(* CODESYS project AlphaController_RECOVERED_2020-08-18T09-54-29.project
   Company: Sharp Packaging
   VersionPostfix: -alpha/pro24
   Version: 0.9.13.2
   Title: MOAB Prototype
   Author: Ben Hess

Project tree, tasks and I/O mapping:
  Device : Advantech Control x86 RTE V3, Advantech Co., Ltd., order no. 
      , version 3.5.13.0
    application Application
      libraries: Standard, * (System); VisuDialogs, * (System); Unit Conversion Interfaces, * (Intern); Festo_Motion_FHPP_3, 3.5.7.21 (Festo AG & Co. KG); Serial Communication, 3.5.7.0 (3S - Smart Software Solutions GmbH); Storage, 3.5.7.0 (3S - Smart Software Solutions GmbH); SysPort, 3.5.5.0 (System); Time and Date, 3.5.7.0 (3S - Smart Software Solutions GmbH); SysTime, 3.5.9.0 (System); Network, 3.5.7.0 (3S - Smart Software Solutions GmbH); CIP Object, * (3S - Smart Software Solutions GmbH); CAA Memory Block Manager Extern, * (CAA Technical Workgroup); CmpBitmapPool, * (System); IoDrvModbusBase, 3.5.13.0 (3S - Smart Software Solutions GmbH); SysFile, 3.5.15.0 (System); SysCom, 3.5.15.0 (System); Recipe Management, 3.5.15.0 (System); IoDrvModbus, 3.5.15.0 (3S - Smart Software Solutions GmbH); SysTypes Interfaces, * (System); BASIC, * (OSCAT)
      task IOUpdate (cyclic, interval 5 ms, priority 1) calls nothing
      task MainTask (cyclic, interval 5 ms, priority 0) calls PRG_MainProgram
      Event Handlers/
        function StartDone [ST]
        function OnlineChangeDone [ST]
        function PrepareShutdown [ST]
        function PrepareOnlineChange [ST]
        function PrepareStop [ST]
      Interfaces/
        interface IFaultHandler: AddActiveFault, RemoveActiveFault
        interface IComponentStatus: Mode, Ready
        interface ISupervisor: NotifyMachineFaulted, MakeReady
      RecipeManager
        recipe definition Recipes: HMIData.initiateCycle : BOOL; HMIData.ackAllFaults : BOOL; HMIData.makeReady : BOOL; HMIData.jobLoaded : BOOL; HMIData.stopMachine : BOOL; HMIData.version : STRING; HMIData.inCycle : BOOL; HMIData.batchEnable : BOOL; HMIData.batchSetting : UDINT; HMIData.batchCount : UDINT; HMIData.headCycleCount : UDINT; HMIData.pressureBarOpenDelay : REAL; HMIData.pressureBarCloseDelay : REAL; HMIData.passthroughSetting : REAL; HMIData.passthroughOffset : REAL; HMIData.passthroughPosition : REAL; HMIData.lpaDwell : REAL; HMIData.hpaDwell : REAL; HMIData.sealBarDwell : REAL; HMIData.sealBarTemperatureSetting : UDINT; HMIData.sealBarTemperature : UDINT; HMIData.sealFlattenersPosition : REAL; HMIData.bagSkirtLength : REAL; HMIData.bagLength : REAL; HMIData.bagWidth : REAL; HMIData.bagThickness : REAL; HMIData.bagTensionSetting : REAL; HMIData.bagDropTime : REAL; HMIData.bagForwardSpeed : UDINT; HMIData.bagReverseSpeed : UDINT; HMIData.bagEdgePhotoeyeCovered : BOOL; HMIData.printSpeed : UDINT; HMIData.printLength : REAL; HMIData.printOffset : REAL; HMIData.fillerCountSetting : UDINT; HMIData.fillerCurrentCount : UDINT; HMIData.fillerDropTime : REAL; HMIData.loadPlateDelay : REAL; HMIData.loadPlateDwell : REAL; HMIData.exitConveyorDwell : REAL; HMIData.vacuumDwell : REAL; HMIData.IBDDeflateDwellTime : REAL; HMIData.IBDPackageEjectAssistDelayTime : REAL; HMIData.IBDPackageEjectAssistDwellTime : REAL; HMIData.funnelInUse : BOOL; HMIData.funnelOpenDelay : REAL; HMIData.funnelOpeningTime : REAL; HMIData.funnelClosingTime : REAL; HMIData.externalExitConveyorDwell : REAL; HMIData.barcodeGoodReadCount : UDINT; HMIData.barcodeBadReadCount : UDINT; HMIData.barcodeBadReadFaultSetting : UDINT; HMIData.barcodeStartPosition : REAL; HMIData.barcodeScanDistance : REAL; HMIData.barcodeVerifierInUse : BOOL; HMIData.barcodeLastReadString : STRING(100); HMIData.lastCycleTime : REAL; HMIData.averageCycleTime : REAL; HMIData.resetAverageCycleTime : BOOL; HMIData.bagOpenRetrySetting : INT; HMIData.bagOpenRetryCount : INT; HMIData.bagOpenFeedNewBagSetting : INT; HMIData.bagOpenFeedNewBagCount : INT; HMIData.currentJobID : INT; HMIData.separateBeforeSeal : BOOL; HMIData.activateDemoMode : BOOL; HMIData.printerInUse : BOOL; HMIData.printerInstalled : BOOL; HMIData.lpaDuringBagFeedEnable : BOOL; HMIData.lpaBagEjectAssistEnable : BOOL; HMIData.lpaServiceOn : BOOL; HMIData.lpaServiceOff : BOOL; HMIData.lpaServicePulse : BOOL; HMIData.hpaServiceOn : BOOL; HMIData.hpaServicePulse : BOOL; HMIData.exitConveyorStart : BOOL; HMIData.exitConveyorStop : BOOL; HMIData.exitConveyorJog : BOOL; HMIData.exitConveyorJogTime : TIME; HMIData.exitConveyorStartDwell : BOOL; HMIData.pressureBarService.extendCommand : BOOL; HMIData.pressureBarService.retractCommand : BOOL; HMIData.pressureBarService.exhaustCommand : BOOL; HMIData.pressureBarService.extendedFeedback : BOOL; HMIData.pressureBarService.retractedFeedback : BOOL; HMIData.loadPlateService.extendCommand : BOOL; HMIData.loadPlateService.retractCommand : BOOL; HMIData.loadPlateService.exhaustCommand : BOOL; HMIData.loadPlateService.extendedFeedback : BOOL; HMIData.loadPlateService.retractedFeedback : BOOL; HMIData.forwardLoadPlateService.extendCommand : BOOL; HMIData.forwardLoadPlateService.retractCommand : BOOL; HMIData.forwardLoadPlateService.exhaustCommand : BOOL; HMIData.forwardLoadPlateService.extendedFeedback : BOOL; HMIData.forwardLoadPlateService.retractedFeedback : BOOL; HMIData.rearLoadPlateService.extendCommand : BOOL; HMIData.rearLoadPlateService.retractCommand : BOOL; HMIData.rearLoadPlateService.exhaustCommand : BOOL; HMIData.rearLoadPlateService.extendedFeedback : BOOL; HMIData.rearLoadPlateService.retractedFeedback : BOOL; HMIData.loadShelfService.extendCommand : BOOL; HMIData.loadShelfService.retractCommand : BOOL; HMIData.loadShelfService.exhaustCommand : BOOL; HMIData.loadShelfService.extendedFeedback : BOOL; HMIData.loadShelfService.retractedFeedback : BOOL; HMIData.IBDService.extendCommand : BOOL; HMIData.IBDService.retractCommand : BOOL; HMIData.IBDService.exhaustCommand : BOOL; HMIData.IBDService.extendedFeedback : BOOL; HMIData.IBDService.retractedFeedback : BOOL; HMIData.funnelService.extendCommand : BOOL; HMIData.funnelService.retractCommand : BOOL; HMIData.funnelService.exhaustCommand : BOOL; HMIData.funnelService.extendedFeedback : BOOL; HMIData.funnelService.retractedFeedback : BOOL; HMIData.jogBagForward : BOOL; HMIData.jogBagReverse : BOOL; HMIData.jogPassthroughForward : BOOL; HMIData.jogPassthroughReverse : BOOL; HMIData.sealBarServiceCycle : BOOL; HMIData.sealBarServiceRetract : BOOL; HMIData.sealBarServiceExtend : BOOL; HMIData.bagOpenFingersServiceGrab : BOOL; HMIData.bagOpenFingersServiceRelease : BOOL; HMIData.sealFlattenersServiceRaise : BOOL; HMIData.sealFlattenersServiceLower : BOOL; HMIData.sealFlattenersServiceJogIn : BOOL; HMIData.sealFlattenersServiceJogOut : BOOL; HMIData.sealFlattenersManualPositionSetting : REAL; HMIData.sealFlattenersMoveToManualPos : BOOL; HMIData.passthroughManualPositionSetting : REAL; HMIData.passthroughMoveToManualPos : BOOL; HMIData.factoryTestMode : BOOL; HMIData.vacuumServiceOn : BOOL; HMIData.vacuumServiceOff : BOOL; HMIData.printHeadServiceRaise : BOOL; HMIData.printHeadServiceLower : BOOL; HMIData.externalExitConveyorStart : BOOL; HMIData.externalExitConveyorStop : BOOL; HMIData.externalExitConveyorJog : BOOL; HMIData.externalExitConveyorStartDwell : BOOL; HMIData.triggerBarcodeReaderService : BOOL; HMIData.bofSelection : INT; HMIData.sealFlattenersSelection : INT; HMIData.printerSelection : INT; HMIData.integratedExitConveyorSelection : INT; HMIData.externalExitConveyorSelection : INT; HMIData.packageEjectSelection : INT; HMIData.independentBagDeflatorSelection : INT; HMIData.cycleStartButtonSelection : INT; HMIData.barcodeVerifierSelection : INT; HMIData.baggerModelSelection : INT; HMIData.auxIOConfig.factorySelection : INT; HMIData.auxIOConfig.cfgInputSelection : INT; HMIData.auxIOConfig.cfgOutput1Selection : INT; HMIData.auxIOConfig.cfgOutput2Selection : INT; HMIData.fillerFactorySelection : INT; HMIData.funnelFactorySelection : INT; HMIData.murrIOConfigVersion : INT; HMIData.printerConfigVersion : INT; HMIData.frontFilmFeedMotorConfigVersion : INT; HMIData.rearUnwindMotorConfigVersion : INT; HMIData.sealFlattenerMotorConfigVersion : INT; HMIData.printerRibbonLow.active : BOOL; HMIData.printerNotReady.active : BOOL; HMIData.waitingForPrinter.active : BOOL; HMIData.sealBarNotAtTemperature.active : BOOL; HMIData.recoveryModeActive.active : BOOL; HMIData.jobLoadRequired.active : BOOL; HMIData.baggerNotReady.active : BOOL; HMIData.demoModeIsActive.active : BOOL; HMIData.factoryTestModeActive.active : BOOL; HMIData.machineNotTested.active : BOOL; HMIData.packageEjectGuardRemoved.active : BOOL; HMIData.bagLevelLow.active : BOOL; HMIData.fillerModeCycleStartOnly.active : BOOL; HMIData.baggerInhibited.active : BOOL; HMIData.pressureBarState : STRING; HMIData.baggerCycles.reset : BOOL; HMIData.baggerCycles.count : UDINT; HMIData.bagOpenFingerCycles.reset : BOOL; HMIData.bagOpenFingerCycles.count : UDINT; HMIData.bagsMade.reset : BOOL; HMIData.bagsMade.count : UDINT; HMIData.sealBarCycles.reset : BOOL; HMIData.sealBarCycles.count : UDINT; HMIData.pressureBarCycles.reset : BOOL; HMIData.pressureBarCycles.count : UDINT; HMIData.passthroughChanges.reset : BOOL; HMIData.passthroughChanges.count : UDINT; HMIData.loadPlateCycles.reset : BOOL; HMIData.loadPlateCycles.count : UDINT; HMIData.printerCycles.reset : BOOL; HMIData.printerCycles.count : UDINT; HMIData.motorizedSealFlattenerCycles.reset : BOOL; HMIData.motorizedSealFlattenerCycles.count : UDINT; HMIData.bagOpenRetryTotal.reset : BOOL; HMIData.bagOpenRetryTotal.count : UDINT; HMIData.bagsRejectedTotal.reset : BOOL; HMIData.bagsRejectedTotal.count : UDINT; HMIData.resettableBagsMade.reset : BOOL; HMIData.resettableBagsMade.count : UDINT; HMIData.airFilterClean.target : UDINT; HMIData.airFilterClean.name : STRING; HMIData.airFilterClean.units : STRING; HMIData.airFilterClean.reset : BOOL; HMIData.airFilterClean.count : UDINT; HMIData.driveRollerClean.target : UDINT; HMIData.driveRollerClean.name : STRING; HMIData.driveRollerClean.units : STRING; HMIData.driveRollerClean.reset : BOOL; HMIData.driveRollerClean.count : UDINT; HMIData.printHeadClean.target : UDINT; HMIData.printHeadClean.name : STRING; HMIData.printHeadClean.units : STRING; HMIData.printHeadClean.reset : BOOL; HMIData.printHeadClean.count : UDINT; HMIData.pressureBarGuideShaftGuides.target : UDINT; HMIData.pressureBarGuideShaftGuides.name : STRING; HMIData.pressureBarGuideShaftGuides.units : STRING; HMIData.pressureBarGuideShaftGuides.reset : BOOL; HMIData.pressureBarGuideShaftGuides.count : UDINT; HMIData.pressureBarLeak.iExtended : BOOL; HMIData.pressureBarLeak.iRetracted : BOOL; HMIData.pressureBarLeak.maximumStrokeTime : REAL; HMIData.pressureBarLeak.strokeTime : REAL; HMIData.pressureBarLeak.strokeTimer.IN : BOOL; HMIData.pressureBarLeak.strokeTimer.PT : TIME; HMIData.pressureBarLeak.strokeTimer.Q : BOOL; HMIData.pressureBarLeak.strokeTimer.ET : TIME; HMIData.pressureBarLeak.extendedONS.CLK : BOOL; HMIData.pressureBarLeak.extendedONS.Q : BOOL; HMIData.pressureBarLeak.retractedONS.CLK : BOOL; HMIData.pressureBarLeak.retractedONS.Q : BOOL; HMIData.pressureBarLeak.target : UDINT; HMIData.pressureBarLeak.name : STRING; HMIData.pressureBarLeak.units : STRING; HMIData.pressureBarLeak.reset : BOOL; HMIData.pressureBarLeak.count : UDINT; HMIData.loadPlateLeak.iExtended : BOOL; HMIData.loadPlateLeak.iRetracted : BOOL; HMIData.loadPlateLeak.maximumStrokeTime : REAL; HMIData.loadPlateLeak.strokeTime : REAL; HMIData.loadPlateLeak.strokeTimer.IN : BOOL; HMIData.loadPlateLeak.strokeTimer.PT : TIME; HMIData.loadPlateLeak.strokeTimer.Q : BOOL; HMIData.loadPlateLeak.strokeTimer.ET : TIME; HMIData.loadPlateLeak.extendedONS.CLK : BOOL; HMIData.loadPlateLeak.extendedONS.Q : BOOL; HMIData.loadPlateLeak.retractedONS.CLK : BOOL; HMIData.loadPlateLeak.retractedONS.Q : BOOL; HMIData.loadPlateLeak.target : UDINT; HMIData.loadPlateLeak.name : STRING; HMIData.loadPlateLeak.units : STRING; HMIData.loadPlateLeak.reset : BOOL; HMIData.loadPlateLeak.count : UDINT; HMIData.msfHorizontalMotorTemp.iDriveTemp : DINT; HMIData.msfHorizontalMotorTemp.maxTemp : REAL; HMIData.msfHorizontalMotorTemp.DriveTemp : REAL; HMIData.msfHorizontalMotorTemp.target : UDINT; HMIData.msfHorizontalMotorTemp.name : STRING; HMIData.msfHorizontalMotorTemp.units : STRING; HMIData.msfHorizontalMotorTemp.reset : BOOL; HMIData.msfHorizontalMotorTemp.count : UDINT; HMIData.bagDeliveryMotorTemp.iDriveTemp : DINT; HMIData.bagDeliveryMotorTemp.maxTemp : REAL; HMIData.bagDeliveryMotorTemp.DriveTemp : REAL; HMIData.bagDeliveryMotorTemp.target : UDINT; HMIData.bagDeliveryMotorTemp.name : STRING; HMIData.bagDeliveryMotorTemp.units : STRING; HMIData.bagDeliveryMotorTemp.reset : BOOL; HMIData.bagDeliveryMotorTemp.count : UDINT; HMIData.passthroughMotorTemp.iDriveTemp : DINT; HMIData.passthroughMotorTemp.maxTemp : REAL; HMIData.passthroughMotorTemp.DriveTemp : REAL; HMIData.passthroughMotorTemp.target : UDINT; HMIData.passthroughMotorTemp.name : STRING; HMIData.passthroughMotorTemp.units : STRING; HMIData.passthroughMotorTemp.reset : BOOL; HMIData.passthroughMotorTemp.count : UDINT; HMIData.faultActive : BOOL
      Types/
        data type DEVICE_MODES
        Factoy Selection/
          data type IntegratedConveyorSelection
          data type LabelPrinterSelection
          data type PackageEjectionSelection
          data type ExteralConveyorSelection
          data type BCVSelection
          data type BagDeflatorSelection
          data type SealFlattenerSelection
          data type PalmButtonSelection
          data type BagOpenFingersSelection
          data type AuxiliaryIOSelection
          data type FillerSelection
          data type ModelSelection
          data type FunnelSelection
        data type MODBUS_COMM_TYPE
        data type LoadPlateFaultsType
        data type MotorCommFault
        data type Fault
        data type QX_PROGRAMS
        data type PRINT_SPEEDS
        States/
          data type SOLENOID_TEST_STATES
          data type AMP_EIP_MOVE_INITIAL_STATES
          data type MOVE_MODBUS_COMMAND_STATES
          data type JOG_STATES
          data type PRESSURE_BAR_STATES
          data type VACUUM_PICKER_STATES
          data type OPCODE_MODBUS_COMMAND_STATES
          data type FILLER_STATES
          data type GRABBER_STATES
          data type BCR_STATES
          data type PASSTHROUGH_SERVO_STATES
          Head/
            data type TEST_HEAD_STATES
            data type PRINTER_STATES
            data type HEAD_STATES
            data type SEAL_FLATTENER_STATES
            data type SEAL_BAR_STATES
            data type SEAL_SEPARATE_STATES
            data type FINISH_CYCLE_STATES
            data type RELEASE_FEED_STATES
            data type BAG_DELIVERY_STATES
            data type BAG_OPEN_ASSIST_STATES
          MurrIOMOdule/
            data type MOM_STATES
            data type MURR_SYSTEM_STATES
          data type JAW_HOMING_STATES
        HMI Types/
          data type PressureBarHMI
        data type ServiceCommands
        data type ORIENTAL_OPERATION_TYPES
        data type PressureBarFaultsType
        data type IOMasterFaultsType
        data type CylinderFaultsType
        data type ModbusLongType
        AuxIO/
          data type AuxOutputSelection
          data type AuxInputSelection
          data type AuxIOConfiguration
        data type Alarm
        data type FaultType
        data type Warning
        data type StepServoFaultsType
        data type STEP_SERVO_OPCODES
        data type CONFIG_VERSIONS
      global variables HMIData
      trace Trace (task MainTask): PRG_Bagger.moabHead.pressureBar.electricPressureBarMotor.CRTL_Axis.AckStart, PRG_Bagger.moabHead.pressureBar.electricPressureBarMotor.CRTL_Axis.StartTask, PRG_Bagger.moabHead.pressureBar.electricPressureBarMotor.CRTL_Axis.ActualRecordNo, PRG_Bagger.moabHead.pressureBar.electricPressureBarMotor.CRTL_Axis.RecordNo
      FBs/
        DataHandlers/
          function block FB_ModbusDWORD [ST]: HighWord, RawValue, LowWord
          function block ModbusLongHandlerFB [ST]: PackDirect, Pack, Unpack
        Fault/
          function block FB_ONS [ST]
          function block FB_GetTime [ST]
          function block FB_Fault [ST]: Execute, InstanceName, RegisterLogger, Ack, Trigger, FB_Init
          data type LogMessageType
          function block FB_HMIFault [ST]: FB_Init, FB_Reinit, Initialize, InstanceName, Execute
          function block FB_InternalLogger [ST]: InstanceName, AddLogItem
        function block FB_TCPClient [ST]: SendLabel
        Cylinders/
          function block FB_CylinderWithFeedback [ST]: Execute
          interface IThreePositonCylinder: Exhaust
          function block FB_CylinderFaults [ST]
          function block FB_Cylinder [ST]: Retract, Extend, Execute
          function block FB_ThreePositionCylinderWithFeedback [ST]: ResetFault, Exhaust, Execute, Faulted
          interface ICylinder: Extend, Execute, Retract
          function block FB_ThreePositionCylinder [ST]: Exhaust
        function block FB_WriteToFile [ST]
        function block FB_PredictiveMaint [ST]
        function block GetTime [ST]
        function block FB_CylinderLeak [ST]
        function block FB_DriveTemp [ST]
        function block TimeLeftFB [ST]
        Components/
          function block PrinterFB_Mode2 [ST]: AutoSendPrintSignal, AutoPrintNow, AutoAckPrintDone, Ready, Mode
          function block BagDeliveryFB_BothMotors [ST]: Ready, ClearCommands, Mode, AutoReverseBag, AutoPrinterDone, AutoWaitForPrinter, AutoStartPrintFeed, AutoFeedBagOut, AutoFeedToEye, AutoPrinterReady
          KeyenceL20FB/
            data type eKeyenceLN20_Error_ID
            function block KeyenceNL20FB [ST]: Ready, Mode
            data type eKeyenceLN20FB_States
          function block MotorizedSealFlattenersFB_BagFeed [ST]: AutoMoveIn, AutoMoveToBagHolding, AutoMoveToHandLoad, Ready, Mode, ClearCommands, AutoMoveToClearance, AutoMoveOut
          function block BarcodeReaderFB [ST]: Trigger, BadRead, GoodRead
          function block BagDeliveryFB [ST]: AutoPrinterDone, AutoFeedToEye, AutoWaitForPrinter, AutoReverseBag, ClearCommands, AutoPrinterReady, Mode, Ready, AutoFeedBagOut, AutoStartPrintFeed
          function block AdjustablePassthroughFB [ST]: MovePassthrough, Ready, Mode, AckRequest, HomeEndStop
          function block FillerFB [ST]: BaggerCycledAndReady, Ready, BaggerCycleInitiated, Mode, Reset
          function block PrinterFB [ST]: AutoSendPrintSignal, AutoPrintNow, Mode, AutoAckPrintDone, Ready
          DelayDwellFB/
            function block DelayDwellFB [ST]: Reset, ManualOff, ManualOn, Trigger, DwellSetting, DelaySetting
            data type DELAY_DWELL_STATES
          FB_MotorizedPressureBar/
            function block FB_CylinderFeedback [ST]
            function block FB_MotorizedPressureBar [ST]: CloseJawNoLatch, CloseJaw, OpenJaw, HomeNow
            data type MotorizedPbarStates
          function block BagOpenFingersFB [ST]: Release, Grab
          function block MotorizedSealFlattenersFB [ST]: ClearCommands, AutoMoveOut, Mode, Ready, AutoMoveToClearance, AutoMoveToBagHolding, AutoMoveIn
          function block PneumaticPressureBarFB_1 [ST]: AutoSealBag, RetractCylinder, AutoOpenJaw, ExhaustCylinder, AutoDoneMovingPassthrough, Mode, ExtendCylinderHighPressure, AutoCloseJaw, Ready, AutoMovingPassthrough, ExtendCylinderLowPressure
          function block FunnelFB [ST]: DelaySetting, CloseNow, OpeningTime, OpenNow, ClosingTime
          FB_MotorizedIBD/
            data type MotorizedIBDStates
            function block FB_MotorizedIBD [ST]: CloseIBD, OpenFull, OpenIBD, RemovePower, HomeNow
          function block PneumaticPressureBarFB [ST]: AutoDoneMovingPassthrough, AutoMovingPassthrough, ExhaustCylinder, Ready, Mode, AutoCloseJaw, ExtendCylinderHighPressure, ExtendCylinderLowPressure, AutoOpenJaw, RetractCylinder, AutoSealBag
          function block ElectricPressureBarFB [ST]: AutoCloseJaw, AutoOpenJaw, Mode, Ready, ClearCommands
          function block PickAndPlaceFB [ST]
          function block BagOpenFingersWithSensorsFB [ST]: CheckIfBagGrabbed
          function block MurrIOFB [ST]: Mode, Ready
          function block BaseComponentFB [ST]: Ready, Reset, Mode
          function block HeadRaiseLowerFB [ST]
          function block MonostableMultivibratorFB [ST]: DelaySetting, Trigger, ManualOn, ManualOff, DwellSetting
        Motors/
          interface IPositionableMotor: Homing, Moving, InPosition, CurrentPosition, Stop, CommandAcknowledged, HomeNow, MoveToPosition, HomeRequired, MoveDistance
          interface IStoredProgramMotor: ActiveStoredProgramNumber, ExecuteStoredProgram
          Applied Motion/
            function block FB_AppliedMotionBagDeliveryMotor_1 [ST]: SetRearMotorToTorqueMode, SetRearMotorToEncoderFollowing, MoveDistance, StopViaProgram, CommandAcknowledged, SetTorque, Execute, SetRearMotorTorqueValue, MoveDistanceFinal
            Modbus Commands/
              function block FB_SendUserRegistersAppliedMotionTCP [ST]: Execute
              function block FB_SendMoveCommandAppliedMotionRTU [ST]: Execute, CheckIfParSendSuccessful
              function block FB_SendBagMoveAppliedMotionTCP [ST]: Execute
              function block FB_SendMoveCommandAppliedMotionTCP [ST]: Execute
              function block FB_SendOpcodeCommandAppliedMotionTCP [ST]: Execute
              function block FB_SendOpcodeCommandAppliedMotionRTU [ST]: Execute
            function block FB_AppliedMotionStepServoMBBase [ST]: Execute, HomeRequired, CommandAcknowledged, ExecuteStoredProgram, ActiveStoredProgramNumber, MoveDistance, InPosition, HomeNow, Stop, Homing, CurrentPosition, Moving, MoveToPosition
            function block FB_AppliedMotionStepServoEIPPassthrough [ST]: HomeNow, DoneClamping, AllowClamping, Stop, SetPositionLimit, Execute
            DataHandlers/
              function block FB_StepServoAlarms [ST]
              function block FB_StepServoCommands [ST]: Enable, AlarmReset, SendHostCommand, FeedToLength, Clear, StopNormal, IdleState, Disable, StopCrash, SendQAndExecute, FeedToPosition
              function block StepServoStatusFB [ST]
            function block FB_AppliedMotionStepServoEIPPassthrough_1 [ST]: DoneClamping, AllowClamping
            function block FB_AppliedMotionBagDeliveryMotorNoFollowing [ST]: MoveDistance, SetRearMotorToTorqueMode, Execute, SetRearMotorToEncoderFollowing, MoveDistanceFinal, CommandAcknowledged, StopViaProgram
            function block FB_AppliedMotionStepServoTCP [ST]: Stop, MoveToPosition, ExecuteStoredProgram, MoveDistance, HomeNow
            function block FB_AppliedMotionStepServoEIPBase [ST]: Stop, Homing, HomeNow, MoveDistance, CommandAcknowledged, InstanceName, MachineFaulted, MoveToPositionTorque, InPosition, Disable, Enable, ResetEncoderPosition, Execute, HomeRequired, ActiveStoredProgramNumber, Reset, Faulted, MoveToPosition, SetTorque, ExecuteStoredProgram, CurrentPosition, Moving, MoveDistanceTorque
            function block FB_AppliedMotionBagDeliveryMotor [ST]: MoveDistance, SendParameters, MoveDistanceFinal, StopViaProgram
            function block FB_AppliedMotionStepServoEIPBaseQX [ST]: Execute, CommandAcknowledged, HomeNow, HomeRequired, Moving, ActiveStoredProgramNumber, InPosition, MoveDistanceTorque, MachineFaulted, Faulted, MoveToPosition, MoveToPositionTorque, Stop, MoveDistance, CurrentPosition, Homing, Reset, RegisterWithFaultHandler, ExecuteStoredProgram
          Festo/
            function block FB_FestoMotor [ST]: ExecuteStoredProgram, Homing, HomeRequired, CurrentPosition, Execute, CommandAcknowledged, Stop, ActiveStoredProgramNumber, InitDrive, Moving, MoveDistance, InPosition, MoveToPosition, HomeNow
        Temp Sensors/
          function block FB_TemperatureSensor [ST]: TempReadingC, TempReadingF, InstanceName
          function block FB_IFMTempSensor [ST]: Execute
          function block FB_TempController [ST]
          interface ITempSensor: TempReadingF, TempReadingC
        function block FB_HMILight [ST]: BlinkSlow, BlinkFast, TurnOff, TurnOn
        function block FB_FaultHandler [ST]: registerFaultSource
        function block SerialMotorTestFB [ST]
        function block FB_BaggerHeadRaise [ST]
        FunctionalAreas/
          function block FB_MOABHead_Electric [ST]
          function block FB_MOABHead [ST]
        function block FB_CycleCounter [ST]: Increment, Clear, SetCount
      Programs/
        program PRG_Bagger [ST]
        program Faults [ST]
        function block PRG_ [ST]
        program PRG_MainProgram [ST]
      global variables Globals
      function SaveValues [ST]
      Symbols
      ObjectHandling/
        interface IExecuteAutomatically: Execute
        function block FB_CollectionHandlerAll [ST]: AddObject
        interface IResettable
        interface IFault: Trigger, Ack
        function block FB_CollectionHandlerLogs [ST]: AddObject
        function block FB_CollectionHandlerLoggable [ST]: RegisterAll, AddObject
        interface IAllObjects: InstanceName
        function block FB_CollectionHandlerInitializable [ST]: InitializeAll, AddObject
        global variables GlobalObjects
        function block FB_CollectionHandlerActiveFaults [ST]: RemoveObject, AckAll, AddObject
        interface ILoggable: RegisterLogger
        interface IInitializable: Initialize
        interface IExhaustable
        interface IFault_1: Ack, Trigger
        function block FB_CollectionHandlerFaults [ST]: AckAll, AddObject
        interface IMachineLogger: AddLogItem
        function block FB_CollectionHandlerExecutable [ST]: ExecuteAll, AddObject
      function RecallValues [ST]
    System_Diagnosis : System Diagnosis, Advantech Co., Ltd., version 3.5.13.0
        unmapped channels: System Information
    CIFX_EIP : CIFX-EIP, 3S - Smart Software Solutions GmbH, order no. 1, version 3.5.12.0
        settings: IPAddress = [16#C0,16#A8,16#0A,16#15]; SubnetMask = [16#FF,16#FF,16#FF,16#00]; GatewayAddress = [16#00,16#00,16#00,16#00]; ConfigVersion = 50660608
      IBD_Motor : SSM23IP-3EG, Applied Motion Products, Inc, order no. SSM23IP-3EG, version Major Revision=16#3, Minor Revision = 16#3
          settings: INITIALIZED = TRUE; IP address of Target = [16#C0,16#A8,16#0A,16#39]; MAC address of Target = [16#00,16#00,16#00,16#00,16#00,16#00]; Keying.Check Device Type = FALSE; Keying.Check Vendor Code = FALSE; Keying.Check Product Code = FALSE; Keying.Check Major Revision = FALSE; Keying.Check Minor Revision = FALSE; RequiredConfigVersion = 50660864; Number of Connections = 1; Connection Settings.Requested packet intervall = 10000 µs; Connection Settings.OT Connection Parameters = 18502; Connection Settings.TO Connection Parameters = 18490; Connection Settings.Connection Flags = 1056; Connection Settings.Connection Path Size = 8; Status Code.ReadOnly = False; Status Code.BitSize = 32; Status Code.DataSize = 4; Alarm Code.ReadOnly = False; Alarm Code.BitSize = 32; Alarm Code.DataSize = 4; Supply Voltage.ReadOnly = False; Supply Voltage.BitSize = 32; Supply Voltage.DataSize = 4; Actual Current.ReadOnly = False; Actual Current.BitSize = 32; Actual Current.DataSize = 4; Drive Temperature.ReadOnly = False; Drive Temperature.BitSize = 32; Drive Temperature.DataSize = 4; Encoder Position.ReadOnly = False; Encoder Position.BitSize = 32; Encoder Position.DataSize = 4; Absolute Position.ReadOnly = False; Absolute Position.BitSize = 32; Absolute Position.DataSize = 4; Position Error.ReadOnly = False; Position Error.BitSize = 32; Position Error.DataSize = 4; Actual Velocity.ReadOnly = False ... (246 more)
          input  iIBDMotorEIP : DINT  // Status Code
          output oIBDMotorEIP : DINT  // Command Word
          unmapped channels: Alarm Code, Supply Voltage, Actual Current, Drive Temperature, Encoder Position, Absolute Position, Position Error, Actual Velocity, Input Status (extended), Input Status (main), Output Status, Analog Input 1 ... (16 more)
      Cube67_BN_E_V2 : Cube67+ BN-E V2, Murrelektronik GmbH, order no. 56535, version Major Revision=16#2, Minor Revision = 16#5
          settings: INITIALIZED = TRUE; IP address of Target = [16#C0,16#A8,16#0A,16#64]; Keying.Check Vendor Code = FALSE; Keying.Check Product Code = FALSE; Keying.Check Major Revision = FALSE; Keying.Check Minor Revision = FALSE; RequiredConfigVersion = 50660864; Number of Connections = 1; Connection Settings.Requested packet intervall = 5000 µs; Connection Settings.OT Connection Parameters = 18624; Connection Settings.TO Connection Parameters = 18708; Connection Settings.Connection Flags = 1056; Connection Settings.Connection Path Size = 8; Input AssemblyParam0.ReadOnly = False; Input AssemblyParam0.BitSize = 8; Input AssemblyParam0.DataSize = 1; Input AssemblyParam1.ReadOnly = False; Input AssemblyParam1.BitSize = 8; Input AssemblyParam1.DataSize = 1; Input AssemblyParam2.ReadOnly = False; Input AssemblyParam2.BitSize = 8; Input AssemblyParam2.DataSize = 1; Input AssemblyParam3.ReadOnly = False; Input AssemblyParam3.BitSize = 8; Input AssemblyParam3.DataSize = 1; Input AssemblyParam4.ReadOnly = False; Input AssemblyParam4.BitSize = 8; Input AssemblyParam4.DataSize = 1; Input AssemblyParam5.ReadOnly = False; Input AssemblyParam5.BitSize = 8; Input AssemblyParam5.DataSize = 1; Input AssemblyParam6.ReadOnly = False; Input AssemblyParam6.BitSize = 8; Input AssemblyParam6.DataSize = 1; Input AssemblyParam7.ReadOnly = False; Input AssemblyParam7.BitSize = 8; Input AssemblyParam7.DataSize = 1; Input AssemblyParam8.ReadOnly = False; Input AssemblyParam8.BitSize = 8; Input AssemblyParam8.DataSize = 1 ... (4114 more)
          input  iAuxFillerTrigger : BOOL  // Input AssemblyParam29.Bit0
          input  iAuxFillerOK : BOOL  // Input AssemblyParam29.Bit1
          input  iAuxConfigInput : BOOL  // Input AssemblyParam29.Bit2
          input  iFunnelOpened : BOOL  // Input AssemblyParam30.Bit0
          input  iRightPalmButton : BOOL  // Input AssemblyParam30.Bit3
          input  iFunnelClosed : BOOL  // Input AssemblyParam31.Bit0
          input  iLeftPalmButton : BOOL  // Input AssemblyParam31.Bit3
          input  iLoadPlateRetracted : BOOL  // Input AssemblyParam32.Bit0
          input  iLoadShelfRetracted : BOOL  // Input AssemblyParam32.Bit1
          input  iEStopOK : BOOL  // Input AssemblyParam32.Bit2
          input  iFrontLoadPlateRetracted : BOOL  // Input AssemblyParam32.Bit3
          input  iHeadLowered : BOOL  // Input AssemblyParam32.Bit6
          input  iLoadPlateExtended : BOOL  // Input AssemblyParam33.Bit0
          input  iLoadShelfExtended : BOOL  // Input AssemblyParam33.Bit1
          input  iFrontLoadPlateExtended : BOOL  // Input AssemblyParam33.Bit3
          input  iBagsLow : BOOL  // Input AssemblyParam33.Bit5
          input  iHeadRaised : BOOL  // Input AssemblyParam33.Bit6
          input  printerDataReady : BOOL  // Input AssemblyParam35.Bit0
          input  printerEndOfPrint : BOOL  // Input AssemblyParam35.Bit1
          input  printerReady : BOOL  // Input AssemblyParam35.Bit2
          input  iPrinterRibbonEncoder : BOOL  // Input AssemblyParam35.Bit3
          input  iBarcodeReadGood : BOOL  // Input AssemblyParam35.Bit4
          input  iJawClampsExtended : BOOL  // Input AssemblyParam36.Bit0
          input  iLefttFingerBagPresent : BOOL  // Input AssemblyParam36.Bit2
          input  iJawClampsRetracted : BOOL  // Input AssemblyParam37.Bit0
          input  iPressureBarNotObstructed : BOOL  // Input AssemblyParam37.Bit1
          input  iRightFingerBagPresent : BOOL  // Input AssemblyParam37.Bit2
          input  iPowerOffButton : BOOL  // Input AssemblyParam37.Bit3
          input  iHeaterBarTempInputs : BYTE  // Input AssemblyParam38
          input  iMurrSystemState : BYTE  // Input Assembly_Param200
          output oMOMConfig : BYTE  // Output AssemblyParam0
          output oAuxBaggerOK : BOOL  // Output Assembly_Param28.Bit0
          output oAuxConfigOut1 : BOOL  // Output Assembly_Param28.Bit1
          output oAuxReadyForFiller : BOOL  // Output Assembly_Param28.Bit2
          output oAuxConfigOut2 : BOOL  // Output Assembly_Param28.Bit3
          output oSoftStart : BOOL  // Output Assembly_Param32.Bit4
          output oBaggerHeadMotorDir : BOOL  // Output Assembly_Param32.Bit7
          output oRunExitConveyor : BOOL  // Output Assembly_Param33.Bit2
          output oRunBaggerHeadMotor : BOOL  // Output Assembly_Param33.Bit7
          output oPrinterStartPrint : BOOL  // Output Assembly_Param34.Bit0
          output oRunPrinterRibbonUnwindMotor : BOOL  // Output Assembly_Param34.Bit1
          output oBarcodeTrigger : BOOL  // Output Assembly_Param34.Bit2
          output oRunExternalExitConveyor : BOOL  // Output Assembly_Param36.Bit1
          output oHMILight : BOOL  // Output Assembly_Param36.Bit3
          output oHeaterPulse : BOOL  // Output Assembly_Param37.Bit4
          unmapped channels: Input AssemblyParam0, Input AssemblyParam1, Input AssemblyParam2, Input AssemblyParam3, Input AssemblyParam4, Input AssemblyParam5, Input AssemblyParam6, Input AssemblyParam7, Input AssemblyParam8, Input AssemblyParam9, Input AssemblyParam10, Input AssemblyParam11 ... (445 more)
      MSFMotor : SSM23IP-3EG, Applied Motion Products, Inc, order no. SSM23IP-3EG, version Major Revision=16#3, Minor Revision = 16#3
          settings: INITIALIZED = TRUE; IP address of Target = [16#C0,16#A8,16#0A,16#35]; Keying.Check Device Type = FALSE; Keying.Check Vendor Code = FALSE; Keying.Check Product Code = FALSE; Keying.Check Major Revision = FALSE; Keying.Check Minor Revision = FALSE; RequiredConfigVersion = 50660864; Number of Connections = 1; Connection Settings.Requested packet intervall = 5000 µs; Connection Settings.OT Connection Parameters = 18502; Connection Settings.TO Connection Parameters = 18490; Connection Settings.Connection Flags = 1056; Connection Settings.Connection Path Size = 8; Status Code.ReadOnly = False; Status Code.BitSize = 32; Status Code.DataSize = 4; Alarm Code.ReadOnly = False; Alarm Code.BitSize = 32; Alarm Code.DataSize = 4; Supply Voltage.ReadOnly = False; Supply Voltage.BitSize = 32; Supply Voltage.DataSize = 4; Actual Current.ReadOnly = False; Actual Current.BitSize = 32; Actual Current.DataSize = 4; Drive Temperature.ReadOnly = False; Drive Temperature.BitSize = 32; Drive Temperature.DataSize = 4; Encoder Position.ReadOnly = False; Encoder Position.BitSize = 32; Encoder Position.DataSize = 4; Absolute Position.ReadOnly = False; Absolute Position.BitSize = 32; Absolute Position.DataSize = 4; Position Error.ReadOnly = False; Position Error.BitSize = 32; Position Error.DataSize = 4; Actual Velocity.ReadOnly = False; Actual Velocity.BitSize = 32 ... (245 more)
          input  sealFlattenerHorizontalMotorInputs : DINT  // Status Code
          output sealFlattenerHorizontalMotorOutputs : DINT  // Command Word
          unmapped channels: Alarm Code, Supply Voltage, Actual Current, Drive Temperature, Encoder Position, Absolute Position, Position Error, Actual Velocity, Input Status (extended), Input Status (main), Output Status, Analog Input 1 ... (16 more)
      Bag_Delivery_Rear_Motor : TSM34IP, Applied Motion Products, Inc, order no. TSM34IP, version Major Revision=16#3, Minor Revision = 16#3
          settings: INITIALIZED = TRUE; IP address of Target = [16#C0,16#A8,16#0A,16#38]; MAC address of Target = [16#00,16#00,16#00,16#00,16#00,16#00]; Keying.Check Device Type = FALSE; Keying.Check Vendor Code = FALSE; Keying.Check Product Code = FALSE; Keying.Check Major Revision = FALSE; Keying.Check Minor Revision = FALSE; RequiredConfigVersion = 50660864; Number of Connections = 1; Connection Settings.Requested packet intervall = 10000 µs; Connection Settings.OT Connection Parameters = 18502; Connection Settings.TO Connection Parameters = 18490; Connection Settings.Connection Flags = 1056; Connection Settings.Connection Path Size = 8; Status Code.ReadOnly = False; Status Code.BitSize = 32; Status Code.DataSize = 4; Alarm Code.ReadOnly = False; Alarm Code.BitSize = 32; Alarm Code.DataSize = 4; Supply Voltage.ReadOnly = False; Supply Voltage.BitSize = 32; Supply Voltage.DataSize = 4; Actual Current.ReadOnly = False; Actual Current.BitSize = 32; Actual Current.DataSize = 4; Drive Temperature.ReadOnly = False; Drive Temperature.BitSize = 32; Drive Temperature.DataSize = 4; Encoder Position.ReadOnly = False; Encoder Position.BitSize = 32; Encoder Position.DataSize = 4; Absolute Position.ReadOnly = False; Absolute Position.BitSize = 32; Absolute Position.DataSize = 4; Position Error.ReadOnly = False; Position Error.BitSize = 32; Position Error.DataSize = 4; Actual Velocity.ReadOnly = False ... (246 more)
          input  bagRearMotorInputs AT %ID200 : DINT  // Status Code
          input  iBagTensionFault : BOOL  // Output Status.Bit3
          output bagRearMotorOutputs AT %QD200 : DINT  // Command Word
          unmapped channels: Alarm Code, Supply Voltage, Actual Current, Drive Temperature, Encoder Position, Absolute Position, Position Error, Actual Velocity, Input Status (extended), Input Status (main), Output Status, Analog Input 1 ... (16 more)
      FestoManifold : CTEU-EP EtherNetIP bus node, Festo AG & Co. KG, order no. CTEU-EP, version Major Revision=16#2, Minor Revision = 16#2
          settings: INITIALIZED = TRUE; IP address of Target = [16#C0,16#A8,16#0A,16#6E]; Keying.Check Vendor Code = FALSE; Keying.Check Product Code = FALSE; Keying.Check Major Revision = FALSE; Keying.Check Minor Revision = FALSE; RequiredConfigVersion = 50660864; Number of Connections = 1; Connection Settings.Requested packet intervall = 10000 µs; Connection Settings.OT Connection Parameters = 18446; Connection Settings.TO Connection Parameters = 18442; Connection Settings.Connection Flags = 1056; Connection Settings.Connection Path Size = 8; Connection Settings.Config#2 Size = 38; Single Port Inputs 8 bytesParam8.ReadOnly = False; Single Port Inputs 8 bytesParam8.BitSize = 8; Single Port Inputs 8 bytesParam8.DataSize = 1; Single Port Inputs 8 bytesParam9.ReadOnly = False; Single Port Inputs 8 bytesParam9.BitSize = 8; Single Port Inputs 8 bytesParam9.DataSize = 1; Single Port Inputs 8 bytesParam10.ReadOnly = False; Single Port Inputs 8 bytesParam10.BitSize = 8; Single Port Inputs 8 bytesParam10.DataSize = 1; Single Port Inputs 8 bytesParam11.ReadOnly = False; Single Port Inputs 8 bytesParam11.BitSize = 8; Single Port Inputs 8 bytesParam11.DataSize = 1; Single Port Inputs 8 bytesParam12.ReadOnly = False; Single Port Inputs 8 bytesParam12.BitSize = 8; Single Port Inputs 8 bytesParam12.DataSize = 1; Single Port Inputs 8 bytesParam13.ReadOnly = False; Single Port Inputs 8 bytesParam13.BitSize = 8; Single Port Inputs 8 bytesParam13.DataSize = 1; Single Port Inputs 8 bytesParam14.ReadOnly = False; Single Port Inputs 8 bytesParam14.BitSize = 8; Single Port Inputs 8 bytesParam14.DataSize = 1; Single Port Inputs 8 bytesParam15.ReadOnly = False; Single Port Inputs 8 bytesParam15.BitSize = 8; Single Port Inputs 8 bytesParam15.DataSize = 1; Single Port Outputs 8bytesParam8.ReadOnly = False; Single Port Outputs 8bytesParam8.BitSize = 8 ... (119 more)
          output oJawClampExtend : BOOL  // Single Port Outputs 8bytesParam8.Bit0
          output oJawClampRetract : BOOL  // Single Port Outputs 8bytesParam8.Bit1
          output oSealBarExtend : BOOL  // Single Port Outputs 8bytesParam8.Bit2
          output oSealBarRetract : BOOL  // Single Port Outputs 8bytesParam8.Bit3
          output oLPAOn : BOOL  // Single Port Outputs 8bytesParam8.Bit4
          output oHPAOn : BOOL  // Single Port Outputs 8bytesParam8.Bit5
          output oLoadPlateExtend : BOOL  // Single Port Outputs 8bytesParam8.Bit6
          output oLoadPlateRetract : BOOL  // Single Port Outputs 8bytesParam8.Bit7
          output oBOFUp : BOOL  // Single Port Outputs 8bytesParam9.Bit0
          output oBOFDown : BOOL  // Single Port Outputs 8bytesParam9.Bit1
          output oPrintHeadDown : BOOL  // Single Port Outputs 8bytesParam9.Bit2
          output oPrintHeadUp : BOOL  // Single Port Outputs 8bytesParam9.Bit3
          output oVacOn : BOOL  // Single Port Outputs 8bytesParam9.Bit4
          output oSealFlatUp : BOOL  // Single Port Outputs 8bytesParam9.Bit6
          output oSealFlatDown : BOOL  // Single Port Outputs 8bytesParam9.Bit7
          output oFrontLoadPlateToLoad : BOOL  // Single Port Outputs 8bytesParam10.Bit2
          output oLoadShelfUp : BOOL  // Single Port Outputs 8bytesParam10.Bit4
          output oIBDExtend : BOOL  // Single Port Outputs 8bytesParam10.Bit6
          output oIBDRetract : BOOL  // Single Port Outputs 8bytesParam10.Bit7
          output oFunnelOpen : BOOL  // Single Port Outputs 8bytesParam11.Bit0
          output oFunnelClose : BOOL  // Single Port Outputs 8bytesParam11.Bit1
          unmapped channels: Single Port Inputs 8 bytesParam8, Single Port Inputs 8 bytesParam9, Single Port Inputs 8 bytesParam10, Single Port Inputs 8 bytesParam11, Single Port Inputs 8 bytesParam12, Single Port Inputs 8 bytesParam13, Single Port Inputs 8 bytesParam14, Single Port Inputs 8 bytesParam15, Single Port Outputs 8bytesParam8, Single Port Outputs 8bytesParam9, Single Port Outputs 8bytesParam10, Single Port Outputs 8bytesParam11 ... (4 more)
      Pbar_ServoEIP : SSM23IP-3EG, Applied Motion Products, Inc, order no. SSM23IP-3EG, version Major Revision=16#3, Minor Revision = 16#3
          settings: INITIALIZED = TRUE; IP address of Target = [16#C0,16#A8,16#0A,16#34]; Keying.Check Vendor Code = FALSE; Keying.Check Product Code = FALSE; Keying.Check Major Revision = FALSE; Keying.Check Minor Revision = FALSE; RequiredConfigVersion = 50660864; Number of Connections = 1; Connection Settings.Requested packet intervall = 5000 µs; Connection Settings.OT Connection Parameters = 18502; Connection Settings.TO Connection Parameters = 18490; Connection Settings.Connection Flags = 1056; Connection Settings.Connection Path Size = 8; Status Code.ReadOnly = False; Status Code.BitSize = 32; Status Code.DataSize = 4; Alarm Code.ReadOnly = False; Alarm Code.BitSize = 32; Alarm Code.DataSize = 4; Supply Voltage.ReadOnly = False; Supply Voltage.BitSize = 32; Supply Voltage.DataSize = 4; Actual Current.ReadOnly = False; Actual Current.BitSize = 32; Actual Current.DataSize = 4; Drive Temperature.ReadOnly = False; Drive Temperature.BitSize = 32; Drive Temperature.DataSize = 4; Encoder Position.ReadOnly = False; Encoder Position.BitSize = 32; Encoder Position.DataSize = 4; Absolute Position.ReadOnly = False; Absolute Position.BitSize = 32; Absolute Position.DataSize = 4; Position Error.ReadOnly = False; Position Error.BitSize = 32; Position Error.DataSize = 4; Actual Velocity.ReadOnly = False; Actual Velocity.BitSize = 32; Actual Velocity.DataSize = 4 ... (244 more)
          input  jawPasstrhoughMotorInputs : DINT  // Status Code
          input  iJawClamped : BOOL  // Input Status (main).Bit1
          input  iJawClearToClamp : BOOL  // Input Status (main).Bit2
          output jawPasstrhoughMotorOutputs : DINT  // Command Word
          unmapped channels: Alarm Code, Supply Voltage, Actual Current, Drive Temperature, Encoder Position, Absolute Position, Position Error, Actual Velocity, Input Status (extended), Input Status (main), Output Status, Analog Input 1 ... (16 more)
      Keyence_BCV : Generic EtherNet/IP device, 3S - Smart Software Solutions GmbH, version 3.5.15.0
          settings: INITIALIZED = TRUE; IP address of Target = [16#C0,16#A8,16#0A,16#A1]; MAC address of Target = [16#00,16#00,16#00,16#00,16#00,16#00]; Keying.Compatibility Bit = FALSE; RequiredConfigVersion = 50660864; Number of Connections = 1; Connection Settings.Requested packet intervall (µs) = 10000; Connection Settings.OT Connection Parameters = 18514; Connection Settings.TO Connection Parameters = 18606; Connection Settings.Connection Flags = 1056; Connection Settings.Connection Path Size = 8; Connection Path = [16#20,16#04,16#24,16#01,16#2C,16#65,16#2C,16#64]; Input_Param0.ReadOnly = False; Input_Param0.BitSize = 8; Input_Param0.DataSize = 1; Input_Param1.ReadOnly = False; Input_Param1.BitSize = 8; Input_Param1.DataSize = 1; Input_Param2.ReadOnly = False; Input_Param2.BitSize = 8; Input_Param2.DataSize = 1; Input_Param3.ReadOnly = False; Input_Param3.BitSize = 8; Input_Param3.DataSize = 1; Input_Param4.ReadOnly = False; Input_Param4.BitSize = 8; Input_Param4.DataSize = 1; Input_Param5.ReadOnly = False; Input_Param5.BitSize = 8; Input_Param5.DataSize = 1; Input_Param6.ReadOnly = False; Input_Param6.BitSize = 8; Input_Param6.DataSize = 1; Input_Param7.ReadOnly = False; Input_Param7.BitSize = 8; Input_Param7.DataSize = 1; Input_Param8.ReadOnly = False; Input_Param8.BitSize = 8; Input_Param8.DataSize = 1; Input_Param9.ReadOnly = False ... (2205 more)
          input  keyenceBCVInputs : BYTE  // Input_Param0
          output keyenceBCVOutputs : BYTE  // Output_Param0
          unmapped channels: Input_Param1, Input_Param2, Input_Param3, Input_Param4, Input_Param5, Input_Param6, Input_Param7, Input_Param8, Input_Param9, Input_Param10, Input_Param11, Input_Param12 ... (234 more)
      Bag_Delivery_EIP_Motor : TSM34IP, Applied Motion Products, Inc, order no. TSM34IP, version Major Revision=16#3, Minor Revision = 16#3
          settings: INITIALIZED = TRUE; IP address of Target = [16#C0,16#A8,16#0A,16#37]; Keying.Check Vendor Code = FALSE; Keying.Check Product Code = FALSE; Keying.Check Major Revision = FALSE; Keying.Check Minor Revision = FALSE; RequiredConfigVersion = 50660864; Number of Connections = 1; Connection Settings.Requested packet intervall = 5000 µs; Connection Settings.OT Connection Parameters = 18502; Connection Settings.TO Connection Parameters = 18490; Connection Settings.Connection Flags = 1056; Connection Settings.Connection Path Size = 8; Status Code.ReadOnly = False; Status Code.BitSize = 32; Status Code.DataSize = 4; Alarm Code.ReadOnly = False; Alarm Code.BitSize = 32; Alarm Code.DataSize = 4; Supply Voltage.ReadOnly = False; Supply Voltage.BitSize = 32; Supply Voltage.DataSize = 4; Actual Current.ReadOnly = False; Actual Current.BitSize = 32; Actual Current.DataSize = 4; Drive Temperature.ReadOnly = False; Drive Temperature.BitSize = 32; Drive Temperature.DataSize = 4; Encoder Position.ReadOnly = False; Encoder Position.BitSize = 32; Encoder Position.DataSize = 4; Absolute Position.ReadOnly = False; Absolute Position.BitSize = 32; Absolute Position.DataSize = 4; Position Error.ReadOnly = False; Position Error.BitSize = 32; Position Error.DataSize = 4; Actual Velocity.ReadOnly = False; Actual Velocity.BitSize = 32; Actual Velocity.DataSize = 4 ... (244 more)
          input  bagDeliveryMotorInputs : DINT  // Status Code
          input  iBagNotPresent : BOOL  // Input Status (main).Bit2
          output bagDeliveryMotorOutputs : DINT  // Command Word
          unmapped channels: Alarm Code, Supply Voltage, Actual Current, Drive Temperature, Encoder Position, Absolute Position, Position Error, Actual Velocity, Input Status (extended), Input Status (main), Output Status, Analog Input 1 ... (16 more)
    Ethernet : Ethernet, 3S - Smart Software Solutions GmbH, version 3.5.15.0
        settings: IPAddress = [192,168,10,20]; SubnetMask = [255,255,255,0]; GatewayAddress = [192,168,10,254]; MACAddress = [16#74,16#FE,16#48,16#3F,16#C0,16#65]; NetworkInterfaceName = 'Machine LAN:2'; NetworkInterfaceName = "Machine LAN:2"; SaveCommunicationSettings = FALSE
      Modbus_TCP_Master : Modbus TCP Master, 3S - Smart Software Solutions GmbH, version 3.5.15.0 (disabled)
          settings: AutoReconnect = TRUE
        Bag_Delivery_Master_Motor : Modbus TCP Slave, 3S - Smart Software Solutions GmbH, version 3.5.15.0 (disabled)
            settings: Unit-ID = 255; IPAddress = [192, 168, 10, 55]; Read Registers.Function Code = 3; Read Registers.Read Offset = 16#0000; Read Registers.Read Length = 125; Read Registers.Write Offset = 0; Read Registers.Write Length = 0; Read Registers.Cycle Time = 50
            input  BagDeliverMasterMotorModbusInputs AT %IW536 : ARRAY[0..124] OF WORD  // Read Registers
        PBar_Servo : Modbus TCP Slave, 3S - Smart Software Solutions GmbH, version 3.5.15.0 (disabled)
            settings: Unit-ID = 255; ResponseTimeout = 100; IPAddress = [192, 168, 10, 52]; Channel 0.Function Code = 3; Channel 0.Read Offset = 16#0000; Channel 0.Read Length = 125; Channel 0.Write Offset = 0; Channel 0.Write Length = 0; Channel 0.Cycle Time = 100
            input  PressureBarEndStopTCPMotorModbusInputs AT %IW800 : ARRAY[0..124] OF WORD  // Channel 0
      EtherNet_IP_Scanner : EtherNet/IP Scanner, 3S - Smart Software Solutions GmbH, order no. 1, version 3.5.15.20
        AMP_Test_Motor : STM23IP-3EN, Applied Motion Products, Inc, order no. STM23IP-3EN, version Major Revision=16#3, Minor Revision = 16#3 (disabled)
            settings: INITIALIZED = TRUE; IP address of Target = [16#C0,16#A8,16#0A,16#37]; Keying.Check Vendor Code = FALSE; Keying.Check Product Code = FALSE; Keying.Check Major Revision = FALSE; Keying.Check Minor Revision = FALSE; RequiredConfigVersion = 50660864; Number of Connections = 1; Connection Settings.Requested packet intervall (µs) = 10000; Connection Settings.OT Connection Parameters = 18502; Connection Settings.TO Connection Parameters = 18490; Connection Settings.Connection Flags = 1056; Connection Settings.Connection Path Size = 8; Connection Path = [16#20,16#04,16#24,16#66,16#2C,16#70,16#2C,16#65]; Status Code.ReadOnly = False; Status Code.BitSize = 32; Status Code.DataSize = 4; Alarm Code.ReadOnly = False; Alarm Code.BitSize = 32; Alarm Code.DataSize = 4; Supply Voltage.ReadOnly = False; Supply Voltage.BitSize = 32; Supply Voltage.DataSize = 4; Actual Current.ReadOnly = False; Actual Current.BitSize = 32; Actual Current.DataSize = 4; Drive Temperature.ReadOnly = False; Drive Temperature.BitSize = 32; Drive Temperature.DataSize = 4; Encoder Position.ReadOnly = False; Encoder Position.BitSize = 32; Encoder Position.DataSize = 4; Absolute Position.ReadOnly = False; Absolute Position.BitSize = 32; Absolute Position.DataSize = 4; Position Error.ReadOnly = False; Position Error.BitSize = 32; Position Error.DataSize = 4; Actual Velocity.ReadOnly = False; Actual Velocity.BitSize = 32 ... (245 more)
            unmapped channels: Status Code, Alarm Code, Supply Voltage, Actual Current, Drive Temperature, Encoder Position, Absolute Position, Position Error, Actual Velocity, Input Status (extended), Input Status (main), Output Status ... (18 more)
        EX260_SEN1 : EX260-SEN1, SMC Corporation, order no. EX260-SEN1, version Major Revision=16#2, Minor Revision = 16#2 (disabled)
            settings: INITIALIZED = TRUE; IP address of Target = [16#C0,16#A8,16#0A,16#A2]; Keying.Check Minor Revision = FALSE; RequiredConfigVersion = 50660864; Number of Connections = 1; Connection Settings.Requested packet intervall (µs) = 20000; Connection Settings.OT Connection Parameters = 18442; Connection Settings.TO Connection Parameters = 18436; Connection Settings.Connection Flags = 1056; Connection Settings.Connection Path Size = 8; Connection Path = [16#20,16#04,16#24,16#69,16#2C,16#96,16#2C,16#64]; Output size.Name = Output size; Output size.ReadOnly = False; Output size.BitSize = 8; Output size.DataSize = 1; Output size.DataType = 'SINT'; Output size.ReadOnly = False; Output size.BitSize = 8; Output size.DataSize = 1; Input size.ReadOnly = False; Input size.BitSize = 16; Input size.DataSize = 1; Output Param0.ReadOnly = False; Output Param0.BitSize = 8; Output Param0.DataSize = 1; Output Param1.ReadOnly = False; Output Param1.BitSize = 8; Output Param1.DataSize = 1; Output Param2.ReadOnly = False; Output Param2.BitSize = 8; Output Param2.DataSize = 1; Output size.ReadOnly = False; Output size.BitSize = 8; Output size.DataSize = 1; Input size.Name = 'Input size'; Input size.HelpString = ''; Input size.ReadOnly = False; Input size.BitSize = 16; Input size.DataSize = 1; Input size.DataType = 'SINT' ... (25 more)
            output oExtendCylinder : BOOL  // Output Param0.Bit0
            output oRetractCylinder : BOOL  // Output Param0.Bit1
            output oExtendSealBar : BOOL  // Output Param0.Bit2
            output oPositionBagOpenFingersToRelease : BOOL  // Output Param0.Bit4
            output oMovePrintHeadDown : BOOL  // Output Param0.Bit6
            unmapped channels: %IB0 Input size, %QB0 Output Param0, %QB1 Output Param1, %QB2 Output Param2, %QB3 Output size
        PickAndPlaceY : STM23IP-3EN, Applied Motion Products, Inc, order no. STM23IP-3EN, version Major Revision=16#2, Minor Revision = 16#33 (disabled)
            settings: INITIALIZED = TRUE; IP address of Target = [16#C0,16#A8,16#0A,16#3B]; Keying.Check Device Type = FALSE; Keying.Check Vendor Code = FALSE; Keying.Check Product Code = FALSE; Keying.Check Major Revision = FALSE; Keying.Check Minor Revision = FALSE; RequiredConfigVersion = 50660864; Number of Connections = 1; Connection Settings.Requested packet intervall (µs) = 50000; Connection Settings.OT Connection Parameters = 18502; Connection Settings.TO Connection Parameters = 18490; Connection Settings.Connection Flags = 1056; Connection Settings.Connection Path Size = 8; Connection Settings.Config#1 Size = 2; Configuration Data = [16#0,16#0]; Connection Path = [16#20,16#04,16#24,16#66,16#2C,16#70,16#2C,16#65]; Status Code.ReadOnly = False; Status Code.BitSize = 32; Status Code.DataSize = 4; Alarm Code.ReadOnly = False; Alarm Code.BitSize = 32; Alarm Code.DataSize = 4; Supply Voltage.ReadOnly = False; Supply Voltage.BitSize = 32; Supply Voltage.DataSize = 4; Actual Current.ReadOnly = False; Actual Current.BitSize = 32; Actual Current.DataSize = 4; Drive Temperature.ReadOnly = False; Drive Temperature.BitSize = 32; Drive Temperature.DataSize = 4; Encoder Position.ReadOnly = False; Encoder Position.BitSize = 32; Encoder Position.DataSize = 4; Absolute Position.ReadOnly = False; Absolute Position.BitSize = 32; Absolute Position.DataSize = 4; Position Error.ReadOnly = False; Position Error.BitSize = 32 ... (248 more)
            input  pickAndPlaceYMotorInputs AT %ID117 : DINT  // Status Code
            output pickAndPlaceYMotorOutputs AT %QD97 : DINT  // Command Word
            unmapped channels: Alarm Code, Supply Voltage, Actual Current, Drive Temperature, Encoder Position, Absolute Position, Position Error, Actual Velocity, Input Status (extended), Input Status (main), Output Status, Analog Input 1 ... (16 more)
        PickAndPlaceX : STM23IP-3EN, Applied Motion Products, Inc, order no. STM23IP-3EN, version Major Revision=16#2, Minor Revision = 16#33 (disabled)
            settings: INITIALIZED = TRUE; IP address of Target = [16#C0,16#A8,16#0A,16#3A]; Keying.Check Device Type = FALSE; Keying.Check Vendor Code = FALSE; Keying.Check Product Code = FALSE; Keying.Check Major Revision = FALSE; Keying.Check Minor Revision = FALSE; RequiredConfigVersion = 50660864; Number of Connections = 1; Connection Settings.Requested packet intervall (µs) = 50000; Connection Settings.OT Connection Parameters = 18502; Connection Settings.TO Connection Parameters = 18490; Connection Settings.Connection Flags = 1056; Connection Settings.Connection Path Size = 8; Connection Settings.Config#1 Size = 2; Configuration Data = [16#0,16#0]; Connection Path = [16#20,16#04,16#24,16#66,16#2C,16#70,16#2C,16#65]; Status Code.ReadOnly = False; Status Code.BitSize = 32; Status Code.DataSize = 4; Alarm Code.ReadOnly = False; Alarm Code.BitSize = 32; Alarm Code.DataSize = 4; Supply Voltage.ReadOnly = False; Supply Voltage.BitSize = 32; Supply Voltage.DataSize = 4; Actual Current.ReadOnly = False; Actual Current.BitSize = 32; Actual Current.DataSize = 4; Drive Temperature.ReadOnly = False; Drive Temperature.BitSize = 32; Drive Temperature.DataSize = 4; Encoder Position.ReadOnly = False; Encoder Position.BitSize = 32; Encoder Position.DataSize = 4; Absolute Position.ReadOnly = False; Absolute Position.BitSize = 32; Absolute Position.DataSize = 4; Position Error.ReadOnly = False; Position Error.BitSize = 32 ... (248 more)
            input  pickAndPlaceXMotorInputs AT %ID103 : DINT  // Status Code
            output pickAndPlaceXMotorOutputs AT %QD81 : DINT  // Command Word
            unmapped channels: Alarm Code, Supply Voltage, Actual Current, Drive Temperature, Encoder Position, Absolute Position, Position Error, Actual Velocity, Input Status (extended), Input Status (main), Output Status, Analog Input 1 ... (16 more)
        PickAndPlaceZ : STM23IP-3EN, Applied Motion Products, Inc, order no. STM23IP-3EN, version Major Revision=16#2, Minor Revision = 16#33 (disabled)
            settings: INITIALIZED = TRUE; IP address of Target = [16#C0,16#A8,16#0A,16#3C]; Keying.Check Device Type = FALSE; Keying.Check Vendor Code = FALSE; Keying.Check Product Code = FALSE; Keying.Check Major Revision = FALSE; Keying.Check Minor Revision = FALSE; RequiredConfigVersion = 50660864; Number of Connections = 1; Connection Settings.Requested packet intervall (µs) = 30000; Connection Settings.OT Connection Parameters = 18502; Connection Settings.TO Connection Parameters = 18490; Connection Settings.Connection Flags = 1056; Connection Settings.Connection Path Size = 8; Connection Settings.Config#1 Size = 2; Configuration Data = [16#0,16#0]; Connection Path = [16#20,16#04,16#24,16#66,16#2C,16#70,16#2C,16#65]; Status Code.ReadOnly = False; Status Code.BitSize = 32; Status Code.DataSize = 4; Alarm Code.ReadOnly = False; Alarm Code.BitSize = 32; Alarm Code.DataSize = 4; Supply Voltage.ReadOnly = False; Supply Voltage.BitSize = 32; Supply Voltage.DataSize = 4; Actual Current.ReadOnly = False; Actual Current.BitSize = 32; Actual Current.DataSize = 4; Drive Temperature.ReadOnly = False; Drive Temperature.BitSize = 32; Drive Temperature.DataSize = 4; Encoder Position.ReadOnly = False; Encoder Position.BitSize = 32; Encoder Position.DataSize = 4; Absolute Position.ReadOnly = False; Absolute Position.BitSize = 32; Absolute Position.DataSize = 4; Position Error.ReadOnly = False; Position Error.BitSize = 32 ... (248 more)
            input  pickAndPlaceZMotorInputs AT %ID1 : DINT  // Status Code
            output pickAndPlaceZMotorOutputs AT %QD113 : DINT  // Command Word
            unmapped channels: Alarm Code, Supply Voltage, Actual Current, Drive Temperature, Encoder Position, Absolute Position, Position Error, Actual Velocity, Input Status (extended), Input Status (main), Output Status, Analog Input 1 ... (16 more)
  Project Information/
    function GetVersion [ST]
    function GetCompany [ST]
    function GetTitle [ST]
    function GetTextProperty2 [ST]
    function GetTextProperty [ST]
    function GetBooleanProperty [ST]
    function GetVersionProperty [ST]
    function GetNumberProperty [ST]
  text list GlobalTextList
  Library Information/
    function IsLibReleased [ST]
    function GetLibVersion [ST]
    function GetLibVersionNumber [ST]
  text list System
*)

// Device/Application/Types/States/Head/TEST_HEAD_STATES
{attribute 'qualified_only'}
{attribute 'strict'}
TYPE TEST_HEAD_STATES :
(
	Idle := 0,
	Cycling := 10,
	StartHoming := 20,
	Homing := 21,
	HomingComplete := 22,
	MovePassthrough := 30,
	MovingPassthrough := 31,
	MovedPassthrough := 32,
	Fault := 99
);
END_TYPE

// Device/Application/Types/DEVICE_MODES
{attribute 'qualified_only'}
{attribute 'strict'}
TYPE DEVICE_MODES :
(
	Manual := 0,	// Control only from service
	Auto := 1,		// Control only from main Bagger Program
	SemiAuto := 2	// Independent control (like as a test fixture)
);
END_TYPE

// Device/Application/Types/States/SOLENOID_TEST_STATES
{attribute 'qualified_only'}
{attribute 'strict'}
TYPE SOLENOID_TEST_STATES :
(
	Extended := 0,
	Retracted := 1,
	FailedToExtend := 2,
	Idle := 3
);
END_TYPE

// Device/Application/Types/Factoy Selection/IntegratedConveyorSelection
{attribute 'qualified_only'}
{attribute 'strict'}
TYPE IntegratedConveyorSelection :
(
	NotInstalled := 0,
	RearExit := 1
);
END_TYPE

// Device/Application/Types/States/Head/PRINTER_STATES
{attribute 'strict'}
{attribute 'qualified_only'}
TYPE PRINTER_STATES :
(
	Idle := 0,
	WaitingForData := 1,
	DataReady := 2,
	BeginPrintCycle := 3,	
	FeedAtPrintSpeed := 10,
	Printing := 11,
	DonePrinting := 20,
	FeedThrough := 21,
	Ready := 40,
	Fault := 99
);
END_TYPE

// Device/Application/Types/Factoy Selection/LabelPrinterSelection
{attribute 'qualified_only'}
{attribute 'strict'}
TYPE LabelPrinterSelection :
(
	NotInstalled := 0,
	ZebraPrinter203DPI := 1,
	ZebraPrinter300DPI := 2
);
END_TYPE

// Device/Application/Types/States/AMP_EIP_MOVE_INITIAL_STATES
{attribute 'strict'}
{attribute 'qualified_only'}
TYPE AMP_EIP_MOVE_INITIAL_STATES :
(
	Idle := 0,
	SetOutputOff := 10,
	WaitAfterSettingOutputOff := 11,
	MoveMotor := 12,
	WaitAfterMovingMotor := 13,
	SetOutputOn := 14,
	WaitAfterSettingOutputOn := 15,
	Fault := 99
);
END_TYPE

// Device/Application/Types/MODBUS_COMM_TYPE
{attribute 'strict'}
{attribute 'qualified_only'}
TYPE MODBUS_COMM_TYPE :
(
	ModbusTCP := 0,
	ModbusRTU := 1
);
END_TYPE

// Device/Application/Types/AuxIO/AuxOutputSelection
{attribute 'qualified_only'}
{attribute 'strict'}
TYPE AuxOutputSelection :
(
	NotConfigured := 0,
	PrinterDataReady := 1,
	WaitingForPrinter := 2,
	CycleComplete := 3,
	BagMade := 4,
	BagMadePlusLabelRequired := 5,
	BagsLow := 6
);
END_TYPE

// Device/Application/Types/LoadPlateFaultsType
TYPE LoadPlateFaultsType :
STRUCT
	failedToDischarge : FB_Fault(name := 'Failed to Discharge');        // Load Plate failed to reach Discharge Position
    failedToLoad : FB_Fault(name := 'Failed to Load');  // Load Plate failed to reach Loading Position
	sensorFault : FB_Fault(name := 'Failed to Sensor Fault');		// Both sensors active at the same time
END_STRUCT
END_TYPE

// Device/Application/Types/States/MOVE_MODBUS_COMMAND_STATES
{attribute 'strict'}
{attribute 'qualified_only'}
TYPE MOVE_MODBUS_COMMAND_STATES :
(
	Idle := 0,
	SendParameters := 10,
	WaitAfterParametersSent := 11,
	SendOpcode := 20,
	WaitAfterOpcodeSent := 21,
	SendCommand := 31,
	WaitAfterCommandSent := 32,
	SendClearCommand := 40,
	WaitAfterSendClearCommand := 41,
	Fault := 99
);
END_TYPE

// Device/Application/Types/MotorCommFault
TYPE MotorCommFault :
STRUCT
	timeOfFault : DATE_AND_TIME;
	message : STRING;
END_STRUCT
END_TYPE

// Device/Application/Types/Factoy Selection/PackageEjectionSelection
{attribute 'qualified_only'}
{attribute 'strict'}
TYPE PackageEjectionSelection :
(
	NotInstalled := 0,
	RearRetractingLoadPlate := 1,
	LabelSideUp := 2
);
END_TYPE

// Device/Application/Types/States/MurrIOMOdule/MOM_STATES
{attribute 'strict'}
{attribute 'qualified_only'}
TYPE MOM_STATES :
(
	Idle := 0,
	Reverse := 1,
	Reversing := 2,
	ReverseToPrinthead := 3,
	ReversingToPrintHead := 4,
	ReverseDone := 5,
	WaitingForPrinter := 10,
	FeedToPrintOffset := 11,
	FeedingToPrintOffset := 12,
	FedToPrintOffset := 13,
	FeedAtPrintSpeed := 20,
	FeedingAtPrintSpeed := 21,
	FedAtPrintSpeed := 22,
	FeedBagOut := 30,
	FeedingBagOut := 31,
	FedBagOut := 32,
	Ready := 40,
	FeedToEye := 50,
	FeedingToEye := 51,
	SetTorqueMode := 52,
	Fault := 99,
	Manual := 100
);
END_TYPE

// Device/Application/Types/States/JOG_STATES
{attribute 'strict'}
{attribute 'qualified_only'}
TYPE JOG_STATES :
(
    Idle := 0,
    JogForwardDIRequest := 10,
    JogForwardOpcodeRequest := 11,
    JoggingForward := 12,
    JogReverseDIRequest := 20,
    JogReverseOpcodeRequest := 21,
    JoggingReverse := 22,
    StoppingJog := 30
);
END_TYPE

// Device/Application/Types/Fault
TYPE Fault :
STRUCT
    name : STRING[20];
    description : STRING[255];
END_STRUCT
END_TYPE

// Device/Application/Types/QX_PROGRAMS
{attribute 'strict'}
TYPE QX_PROGRAMS :
(
    HOME_HARD_STOP := 1
);
END_TYPE

// Device/Application/Types/Factoy Selection/ExteralConveyorSelection
{attribute 'qualified_only'}
{attribute 'strict'}
TYPE ExteralConveyorSelection :
(
	NotInstalled := 0,
	ExternalExitConveyor := 1
);
END_TYPE

// Device/Application/Types/PRINT_SPEEDS
{attribute 'qualified_only'}
{attribute 'strict'}
TYPE PRINT_SPEEDS :
(
	Two_IPS := 2
);
END_TYPE

// Device/Application/Types/States/PRESSURE_BAR_STATES
{attribute 'strict'}
{attribute 'qualified_only'}
TYPE PRESSURE_BAR_STATES :
(
	Idle := 0,
	OpenJaw := 10,
	OpeningJaw := 11,
	JawOpened := 12,
	CloseJaw := 20,
	ClosingJaw := 21,
	JawClosed := 22,
	Sealing := 30,
	Manual := 40,
	Homing := 41,
	Fault := 99
);
END_TYPE

// Device/Application/Types/Factoy Selection/BCVSelection
{attribute 'qualified_only'}
{attribute 'strict'}
TYPE BCVSelection :
(
	NotInstalled := 0,
	VisionBased := 1,
	LaserScanner := 2,
	TwoDimensional := 3
);
END_TYPE

// Device/Application/Types/States/MurrIOMOdule/MURR_SYSTEM_STATES
{attribute 'qualified_only'}
TYPE MURR_SYSTEM_STATES :
(
	Internal_Comm_OK := 1,
	Waiting_For_MOM := 2,
	Configuring_MOM := 4,
	Internal_Comm_Disabled := 8,
	No_Comm_To_Configured_Node := 127
);
END_TYPE

// Device/Application/Types/States/Head/HEAD_STATES
{attribute 'qualified_only'}
{attribute 'strict'}
TYPE HEAD_STATES :
(
	Idle := 0,
	SealAndSeparateBag := 10,
	SealingAndSeparatingBag := 11,
	SealedAndSeparatedBag := 12,
	ReleaseAndFeedBag := 20,
	ReleasingAndFeedingBag := 21,
	ReleasedAndFedBag := 22,
	OpenBag := 30,
	OpeningBag := 31,
	OpenedBag := 32,
	FinishCycle := 40, 
	FinishingCycle := 41,
	FinishedCycle := 42,
	StartReset := 50,
	Resetting := 51,
	StartHoming := 53,
	Homing := 54,
	HomingComplete := 55,
	MovePassthrough := 60,
	MovingPassthrough := 61,
	MovedPassthrough := 62,
	Fault := 99
);
END_TYPE

// Device/Application/Types/States/Head/SEAL_FLATTENER_STATES
{attribute 'strict'}
{attribute 'qualified_only'}
TYPE SEAL_FLATTENER_STATES :
(
	Idle := 0,
	MoveFlattenersOut := 10,
	MovingFlattenersOut := 11,
	MovedFlattenersOut := 12,
	MoveFlattenersUpAndToClearance := 20,
	MovingFlattenersUpAndToClearance := 21,
	MovedFlattenersUpAndToClearance := 22,
	MoveFlattenersToBagFeed := 23,
	MovingFlattenersToBagFeed := 24,
	MovedFlattenersToBagFeed := 25,
	MoveFlattenersIn := 30,
	MovingFlattenersIn := 31,
	MovedFlattenersIn := 32,
	MoveFlattenersDown := 40,
	MovingFlattenersDown := 41,
	MovedFlattenersDown := 42,
	MoveFlattenersToBagHolding := 50,
	MovingFlattenersToBagHolding := 51,
	MovedFlattenersToBagHolding := 52,
	Ready := 60,
	Fault := 99
);
END_TYPE

// Device/Application/Types/Factoy Selection/BagDeflatorSelection
{attribute 'qualified_only'}
{attribute 'strict'}
TYPE BagDeflatorSelection :
(
	NotInstalled := 0,
	IBDStandard := 1,
	IBDWithHingedPlate := 2,
	MotorizedIBD := 3
);
END_TYPE

// Device/Application/Types/States/Head/SEAL_BAR_STATES
{attribute 'strict'}
{attribute 'qualified_only'}
TYPE SEAL_BAR_STATES :
(
	Idle := 0,
	ExtendSealBar := 10,
	ExtendingSealBar := 11,
	SealBarExtened := 12,
	RetractSealBar := 20,
	RetractingSealBar := 21,
	RetractedSealBar := 22,
	Fault := 99
);
END_TYPE

// Device/Application/Types/States/Head/SEAL_SEPARATE_STATES
{attribute 'qualified_only'}
{attribute 'strict'}
TYPE SEAL_SEPARATE_STATES :
(
	Idle := 0,
	BringInIBD := 8,
	WaitForJawCloseDelay := 9,
	MoveJawIn := 10,
	MovingJawIn := 11,
	MovedJawIn := 12,
	ReverseBag := 20,
	ReversingBag := 21,
	ReversedBag := 22,
	SealBag := 30, 
	SealingBag := 31, 
	SealedBag := 32,
	Done := 100,
	Fault := 99
);
END_TYPE

// Device/Application/Types/ServiceCommands
TYPE ServiceCommands : 
STRUCT
	extendCommand : BOOL;
	retractCommand : BOOL;
	exhaustCommand : BOOL;
	extendedFeedback : BOOL;
	retractedFeedback : BOOL;
END_STRUCT
END_TYPE

// Device/Application/Types/States/VACUUM_PICKER_STATES
{attribute 'strict'}
{attribute 'qualified_only'}
TYPE VACUUM_PICKER_STATES :
(
	Idle := 0,
	Home := 1, 
	Homing := 2, 
	Homed := 3,
	XAxisMoveIn := 10,
	XAxisMovingIn := 11, 
	XaxisMovedIn := 12,
	VacuumTurnOn := 20,
	VacuumHeadDown := 30,
	YAxisMoveDown := 31,
	VacuumHeadAndYAxisMovingDown := 32,
	VacuumHeadAndYAxisMovedDown := 33,
	VacuumTurnOff := 40,
	ConveyorTurnOn := 50,
	ConveyorMoving := 51,
	ConveyorDone := 52,

	Fault := 99,
	Ready := 100,
	Manual := 101
);
END_TYPE

// Device/Application/FBs/Components/FB_MotorizedIBD/MotorizedIBDStates
{attribute 'qualified_only'}
{attribute 'strict'}
TYPE MotorizedIBDStates :
(
	Idle := 0,
	Homing := 9,
	Initialize := 10,
	Initializing := 11,
	Initialized := 12,
	MoveJawOut := 20,
	MovingJawOut := 21,
	MovedJawOut := 22,
	MoveJawIn := 30,
	MovingJawIn := 31,
	MovedJawIn := 32,
	StartClamping := 40,
	StartedClamping := 41,
	Clamping := 42, 
	ReleaseClamp := 43, 
	ReleasingClamp := 44,
	MoveOutFull := 50,
	MovingOutFull := 51,
	MovedOutFull := 52,
	Faulting := 98,
	Faulted := 99
);
END_TYPE

// Device/Application/FBs/Components/DelayDwellFB/DELAY_DWELL_STATES
{attribute 'qualified_only'}
{attribute 'strict'}
TYPE DELAY_DWELL_STATES :
(
	Idle := 0,
	Delay := 1,
	Dwell := 2,
	ResettingDwell := 10,
	ManualOn := 20,
	ManualOff := 21
);
END_TYPE

// Device/Application/Types/Factoy Selection/SealFlattenerSelection
{attribute 'qualified_only'}
{attribute 'strict'}
TYPE SealFlattenerSelection :
(
	NotInstalled := 0,
	MotorizedSealFlatteners := 1
);
END_TYPE

// Device/Application/Types/States/OPCODE_MODBUS_COMMAND_STATES
{attribute 'strict'}
{attribute 'qualified_only'}
TYPE OPCODE_MODBUS_COMMAND_STATES :
(
	Idle := 0,
	SendOpcodeAndParameters := 10,
	WaitAfterOpcodeAndParametersSent := 11,
	Fault := 99
);
END_TYPE

// Device/Application/Types/States/FILLER_STATES
{attribute 'strict'}
{attribute 'qualified_only'}
TYPE FILLER_STATES :
(
	Idle := 0,
	CycleBaggerToActiveFiller := 10,
	WaitingForFiller := 11,
	Dropping := 13,
	BaggerCycling := 14,
	Fault := 99
);
END_TYPE

// Device/Application/Types/States/Head/FINISH_CYCLE_STATES
{attribute 'qualified_only'}
{attribute 'strict'}
TYPE FINISH_CYCLE_STATES :
(
	Idle := 0,
	Start := 1,
	OpenFunnel := 10, 
	OpeningFunnel := 11, 
	OpenedFunnel := 12,
	ClosingFunnelForRetry := 13,
	FunnelClosed := 14,
	BringSealFlattenersInAndDown := 20, 
	BringingSealFlattenersInAndDown := 21,
	SealFlattenersInAndDown := 22,
	BringSealFlattenersToBagHolding := 30,
	BringingSealFlattenersToBagHolding := 31,
	SealFlattenersAtBagHolding := 32,
	Done := 100,
	Fault := 99
);
END_TYPE

// Device/Application/Types/States/GRABBER_STATES
{attribute 'strict'}
{attribute 'qualified_only'}
TYPE GRABBER_STATES :
(
	Idle := 0,
	OpenGrippers := 10,
	MoveGrippersOut := 11,
	MovingGrippersOut := 12,
	GrippersMovedOut :=13,
	MoveGantryUp := 20,
	MovingGantryUp := 21,
	GantryMovedUp := 22,
	MoveGrippersIn := 30,
	MovingGrippersIn := 31,
	GrippersMovedIn := 32,
	Ready := 40,
	GrabBag := 50,
	MoveGantryDown := 60,
	MovingGantryDown := 61,
	GantryMovedDown := 62,
	ReleaseBag := 70,
	Fault := 99
);
END_TYPE

// Device/Application/Types/Factoy Selection/PalmButtonSelection
{attribute 'qualified_only'}
{attribute 'strict'}
TYPE PalmButtonSelection :
(
	NotInstalled := 0,
	SinglePalmButton := 1,
	DualPalmButton := 2
);
END_TYPE

// Device/Application/FBs/Fault/LogMessageType
TYPE LogMessageType :
STRUCT
	logTime : DATE_AND_TIME;
	logMessage : STRING;
END_STRUCT
END_TYPE

// Device/Application/Types/ORIENTAL_OPERATION_TYPES
{attribute 'qualified_only'}
{attribute 'strict'}
TYPE ORIENTAL_OPERATION_TYPES :
(
    NoSetting := 0,
    AbsolutePositioning := 1,
    IncrementalPositioning := 2
);
END_TYPE

// Device/Application/FBs/Components/KeyenceL20FB/eKeyenceLN20_Error_ID
{attribute 'qualified_only'}
{attribute 'strict'}
TYPE eKeyenceLN20_Error_ID :
(
	NO_ERROR := 0,
	OPERATION_INSTRUCTION_ERROR := 120,
	BANK_NUMBER_ERROR := 102,
	EIP_UPDATE_ERROR := 230
);
END_TYPE

// Device/Application/FBs/Components/FB_MotorizedPressureBar/MotorizedPbarStates
{attribute 'qualified_only'}
{attribute 'strict'}
TYPE MotorizedPbarStates :
(
	Idle := 0,
	Homing := 9,
	Initialize := 10,
	Initializing := 11,
	Initialized := 12,
	MoveJawOut := 20,
	MovingJawOut := 21,
	MovedJawOut := 22,
	MoveJawIn := 30,
	MovingJawIn := 31,
	MovedJawIn := 32,
	StartClamping := 40,
	StartedClamping := 41,
	Clamping := 42, 
	ReleaseClamp := 43, 
	ReleasingClamp := 44,
	Faulting := 98,
	Faulted := 99
);
END_TYPE

// Device/Application/Types/States/BCR_STATES
{attribute 'strict'}
{attribute 'qualified_only'}
TYPE BCR_STATES :
(
	Idle := 0,
	WaitForOffset := 10,
	TriggerReader := 11,
	WaitingForResult := 12,
	Resetting := 13
);
END_TYPE

// Device/Application/Types/PressureBarFaultsType
TYPE PressureBarFaultsType :
STRUCT
	failedToOpen : FB_Fault(name := 'Pressure Bar Failed to Open');        // Pressure Bar was commanded to extend but failed to reach the sensor
    failedToClose : FB_Fault(name := 'Pressure Bar Failed to Close');      // Pressure Bar was commanded to retract but failed to reach the sensor
	sensorFault : FB_Fault(name := 'Pressure Bar Sensor Fault');		// Both the open and close sensors active at the same time
	obstructionDetected : FB_Fault(name := 'Pressure Bar Obstruction Detected');		// Pressure Bar detected an obstruction
	obstructionFailedToSwitch : FB_Fault(name := 'Pressure Bar Obstruction Detected'); // Pressure bar obstruction sensors should switch when closed
END_STRUCT
END_TYPE

// Device/Application/Types/Factoy Selection/BagOpenFingersSelection
{attribute 'qualified_only'}
{attribute 'strict'}
TYPE BagOpenFingersSelection :
(
	NotInstalled := 0,
	PneumaticWithBagOpenSensors := 1
);
END_TYPE

// Device/Application/Types/HMI Types/PressureBarHMI
TYPE PressureBarHMI :
STRUCT
	openDelay : UINT;
	closeDelay : UINT;
	passthroughSetting : REAL;
	lowPressureAirDwell : REAL;
	highPressureAirDwell : REAL;
END_STRUCT
END_TYPE

// Device/Application/Types/AuxIO/AuxInputSelection
{attribute 'qualified_only'}
{attribute 'strict'}
TYPE AuxInputSelection :
(
	NotConfigured := 0,
	BaggerInhibit := 1
);
END_TYPE

// Device/Application/Types/States/Head/RELEASE_FEED_STATES
{attribute 'qualified_only'}
{attribute 'strict'}
TYPE RELEASE_FEED_STATES :
(
	Idle := 0,
	MoveJawOutAndDropBag := 10,
	MovingJawOutAndDroppingBag := 11,
	MovingJawOutAndFeedBag := 12,
	MovingJawOutAndFeedingBag := 13,
	MovedJawOutAndFedBag := 15,
	WaitForPrinter := 20,
	FeedToOffset := 21,
	FeedingToOffset := 22,
	StartPrinting := 23,
	SendPrintSignal := 24,
	Printing := 25, 
	StopPrinting := 26,
	Done := 100,
	Fault := 99
);
END_TYPE

// Device/Application/Types/IOMasterFaultsType
TYPE IOMasterFaultsType :
STRUCT
	commFail : FB_Fault(name := 'Communication Fail');	// IO Master to Controller Communication Failure
END_STRUCT
END_TYPE

// Device/Application/Types/CylinderFaultsType
TYPE CylinderFaultsType :
STRUCT
	failedToExtend : FaultType;        // Cylinder was commanded to extend but failed to reach the sensor
    failedToRetract : FaultType;      // Cylinder was commanded to retract but failed to reach the sensor
	sensorFault : FaultType;		// Both Extend and Retract sensors active at the same time
END_STRUCT
END_TYPE

// Device/Application/Types/ModbusLongType
TYPE ModbusLongType :
STRUCT
    highWord : WORD;
    lowWord : WORD;
    displayValue : DINT;
    rawValue : DINT;
END_STRUCT
END_TYPE

// Device/Application/Types/Alarm
TYPE Alarm :
STRUCT
	active : BOOL;
	acknowledged : BOOL;
	ackCommand : BOOL;
END_STRUCT
END_TYPE

// Device/Application/Types/Factoy Selection/AuxiliaryIOSelection
{attribute 'qualified_only'}
{attribute 'strict'}
TYPE AuxiliaryIOSelection :
(
	NotInstalled := 0,
	AuxIOStandard := 1
);
END_TYPE

// Device/Application/Types/States/PASSTHROUGH_SERVO_STATES
{attribute 'strict'}
{attribute 'qualified_only'}
TYPE PASSTHROUGH_SERVO_STATES :
(
	Idle := 0,
	HomingRequired := 1,
	StartHoming := 10,
	Homing := 11,
	HomeComplete := 12,
	MovePassthroughOut := 20,
	MovingPassthroughOut := 21,
	PassthroughMovedOut := 22,
	MovePassthroughIn := 30,
	MovingPassthroughIn := 31,
	PassthroughMovedIn := 32,
	Ready := 40,
	Fault := 99
);
END_TYPE

// Device/Application/Types/States/Head/BAG_DELIVERY_STATES
{attribute 'strict'}
{attribute 'qualified_only'}
TYPE BAG_DELIVERY_STATES :
(
	Idle := 0,
	Reverse := 1,
	Reversing := 2,
	ReverseToPrinthead := 3,
	ReversingToPrintHead := 4,
	ReverseDone := 5,
	WaitingForPrinter := 10,
	FeedToPrintOffset := 11,
	FeedingToPrintOffset := 12,
	FedToPrintOffset := 13,
	FeedAtPrintSpeed := 20,
	FeedingAtPrintSpeed := 21,
	FedAtPrintSpeed := 22,
	FeedBagOut := 30,
	FeedingBagOut := 31,
	FedBagOut := 32,
	Ready := 40,
	FeedToEye := 50,
	FeedingToEye := 51,
	SetTorqueMode := 52,
	Fault := 99,
	Manual := 100
);
END_TYPE

// Device/Application/Types/AuxIO/AuxIOConfiguration
TYPE AuxIOConfiguration :
STRUCT
	factorySelection : AuxiliaryIOSelection;
	cfgInputSelection : AuxInputSelection;
	cfgOutput1Selection : AuxOutputSelection;
	cfgOutput2Selection : AuxOutputSelection;
END_STRUCT
END_TYPE

// Device/Application/Types/FaultType
TYPE FaultType :
STRUCT
	active : BOOL;
	acknowledged : BOOL;
	ackCommand : BOOL;
END_STRUCT
END_TYPE

// Device/Application/FBs/Components/KeyenceL20FB/eKeyenceLN20FB_States
{attribute 'qualified_only'}
{attribute 'strict'}
TYPE eKeyenceLN20FB_States :
(
	Idle := 0,
	WaitForStatus := 2,
	SetStatus := 3,
	WaitForReadClear := 4,
	Reset := 100
);
END_TYPE

// Device/Application/Types/Warning
TYPE Warning :
STRUCT
	active : BOOL;
END_STRUCT
END_TYPE

// Device/Application/Types/StepServoFaultsType
TYPE StepServoFaultsType :
STRUCT
	positionLimit : FB_Fault(name := 'Motor exceeded position limit - following error');        // Motor exceeded position limit - following error
	CCWLimit : FB_Fault(name := 'Counter-Clockwise Limit Reached'); // Counter-Clockwise Limit Reached
	CWLimit : FB_Fault(name := 'Clockwise Limit Reached');		// Clockwise Limit Reached
    overTemp : FB_Fault(name := 'Motor Over Temperature Limit');      // Motor Over Temperature Limit
    internalVoltage : FB_Fault(name := 'Internal Voltage Fault');      // Internal Voltage Fault
    overVoltage    : FB_Fault(name := 'Overvoltage Fault');      // Overvoltage Fault
	underVoltage : FB_Fault(name := 'Undervoltage Fault'); 	// Undervoltage Fault
    overCurrent : FB_Fault(name := 'Motor Overcurrent');      // Motor Overcurrent
    openMotorWinding : FB_Fault(name := 'Motor Detected Open Winding');      // Motor Detected Open Winding
    badEncoder : FB_Fault(name := 'Motor Encoder Failure');      // Motor Encoder Failure
	noMove : FB_Fault(name := 'No Move After Command');
	currentFoldback : FB_Fault(name := 'Current Foldback');
	commFail : FB_Fault(name := 'Drive to Controller Communication Failure');	// Drive to Controller Communication Failure
	notHomed : FB_Fault(name := 'Drive is not homed'); // Drive is not homed
END_STRUCT
END_TYPE

// Device/Application/Types/Factoy Selection/FillerSelection
{attribute 'qualified_only'}
{attribute 'strict'}
TYPE FillerSelection :
(
	NotInstalled := 0,
	StandardFiller := 1
);
END_TYPE

// Device/Application/Types/Factoy Selection/ModelSelection
{attribute 'qualified_only'}
{attribute 'strict'}
TYPE ModelSelection :
(
	Pro18 := 0,
	Pro24 := 1
);
END_TYPE

// Device/Application/Types/STEP_SERVO_OPCODES
{attribute 'strict'}
{attribute 'qualified_only'}
//Taken from Host-Command-Reference pdf on Applied Motion website
TYPE STEP_SERVO_OPCODES :
(
	ALARM_RESET := 16#BA,     
	START_JOGGING := 16#96,     
	STOP_JOGGING := 16#D8,     
	ENCODER_FUNCTION := 16#D6,     //0
	ENCODER_POSITION := 16#98,     //Position
	FEED_TO_DOUBLE_SENSOR := 16#69,     //I/O Point 1 Condition 1 I/O Point 2 Condition 2
	FOLLOW_ENCODER := 16#CC,     //I/O Point Condition
	FEED_TO_LENGTH := 16#66,     
	FEED_TO_SENSOR_WITH_MASK_DISTANCE := 16#6A,     //I/O Point Condition
	FEED_AND_SET_OUTPUT := 16#68,     //I/O Point Condition
	FEED_TO_POSITION := 16#67,     
	FEED_TO_SENSOR := 16#6B,     //I/O Point Condition
	FEED_TO_SENSOR_WITH_SAFETY_DISTANCE := 16#6C,     //I/O Point Condition
	JOG_DISABLE := 16#A3,     
	JOG_ENABLE := 16#A2,     
	MOTOR_DISABLE := 16#9E,     
	MOTOR_ENABLE := 16#9F,     
	SEEK_HOME := 16#6E,     //I/O Point Condition
	SET_POSITION := 16#A5,     //Position
	FILTER_INPUT := 16#C0,     //I/O Point Filter Time
	FILTER_SELECT_INPUTS := 16#D3,     
	STEP_FILTER_FREQ := 16#06,     //Freq
	ANALOG_DEADBAND := 16#D2,     //0.001 V
	ALARM_RESET_INPUT := 16#46,     //Function ('1'..'3') I/O Point
	ALARM_OUTPUT := 16#47,     //Function ('1'..'3') I/O Point
	ANALOG_SCALING := 16#D1,     
	DEFINE_LIMITS := 16#42,     //1..3
	SET_OUTPUT := 16#8B,     //I/O Point Condition
	WAIT_FOR_INPUT := 16#70,     
	QUEUE_LOAD_AND_EXECUTE := 16#78,     //1..12
	WAIT_TIME := 16#6F,     //0.01 sec
	STOP_MOVE_KILL_BUFFER := 16#E1,    
	STOP_MOVE_KILL_BUFFER_NORMAL_DECEL := 16#E2,
	STOP_MOVE := 16#B5  // Might work, might not     
);
END_TYPE

// Device/Application/Types/Factoy Selection/FunnelSelection
{attribute 'qualified_only'}
{attribute 'strict'}
TYPE FunnelSelection :
(
	NotInstalled := 0,
	FunnelWithSensors := 1,
	FunnelWithoutSensors := 2
);
END_TYPE

// Device/Application/Types/CONFIG_VERSIONS
{attribute 'strict'}
{attribute 'qualified_only'}
TYPE CONFIG_VERSIONS :
(
	V_1_0,
	V_1_1,
	V_1_2,
	V_1_3,
	V_1_4,
	V_1_5,
	V_1_6,
	V_1_7,
	V_1_8,
	V_1_9,
	V_1_10,
	V_1_11,
	V_1_12,
	V_1_13,
	V_1_14,
	V_1_15,
	V_1_16,
	V_1_17,
	V_1_18,
	V_1_19,
	V_1_20,
	V_1_21,
	V_1_22,
	V_1_23,
	V_1_24,
	V_1_25,
	V_1_26,
	V_1_27,
	V_1_28,
	V_1_29,
	V_1_30,
	V_1_31,
	V_1_32,
	V_1_33,
	V_1_34,
	V_1_35,
	V_1_36,
	V_1_37,
	V_1_38,
	V_1_39,
	V_1_40,
	V_1_41,
	V_1_42,
	V_1_43,
	V_1_44,
	V_1_45,
	V_1_46,
	V_1_47,
	V_1_48,
	V_1_49,
	V_2_0,
	V_2_1,
	V_2_2,
	V_2_3,
	V_2_4,
	V_2_5,
	V_2_6,
	V_2_7,
	V_2_8,
	V_2_9,
	V_2_10,
	V_2_11,
	V_2_12,
	V_2_13,
	V_2_14,
	V_2_15,
	V_2_16,
	V_2_17,
	V_2_18,
	V_2_19,
	V_2_20,
	V_2_21,
	V_2_22,
	V_2_23,
	V_2_24,
	V_2_25,
	V_2_26,
	V_2_27,
	V_2_28,
	V_2_29,
	V_2_30,
	V_2_31,
	V_2_32,
	V_2_33,
	V_2_34,
	V_2_35,
	V_2_36,
	V_2_37,
	V_2_38,
	V_2_39,
	V_2_40,
	V_2_41,
	V_2_42,
	V_2_43,
	V_2_44,
	V_2_45,
	V_2_46,
	V_2_47,
	V_2_48,
	V_2_49
);
END_TYPE

// Device/Application/Types/States/JAW_HOMING_STATES
{attribute 'strict'}
{attribute 'qualified_only'}
TYPE JAW_HOMING_STATES :
(
    Idle := 0,
    MoveForwardFromSensor := 10,
    MovingForwardFromSensor := 11,
	ClearToHome := 12,
    StartHoming := 13,
    Homing := 14,
    HomeComplete := 15,
	MoveToTwoInches := 16, 
	MovingToTwoInches := 17,
	SetLimits := 18
	
);
END_TYPE

// Device/Application/Types/States/Head/BAG_OPEN_ASSIST_STATES
{attribute 'qualified_only'}
{attribute 'strict'}
TYPE BAG_OPEN_ASSIST_STATES :
(
	Idle := 0,
	MoveJawIn := 10,
	MovingJawIn := 11,
	MovedJawIn := 12,
	MoveJawOut := 20,
	MovingJawOutAndGrab := 21,
	CheckForSuccessfulBagGrab := 22,
	BagFailedToOpen := 23,
	BagOpened := 24,
	MovingJawOutAfterGrab := 25,
	MovedJawOut := 26,
	FeedNewBag := 27,
	Done := 100,
	Fault := 99
);
END_TYPE

// Device/Application/HMIData
// All HMI data is presented through this GVL
{attribute 'qualified_only'}
{attribute 'global_init_slot' := '50001'}
VAR_GLOBAL //PERSISTENT RETAIN
	initiateCycle : BOOL;  // Initiate Cycle Pushbutton
	ackAllFaults : BOOL; // Acknowledge All Faults from HMI
	makeReady : BOOL;
	jobLoaded : BOOL;
    stopMachine : BOOL;
	version : STRING;
	inCycle : BOOL;
	batchEnable : BOOL;
	batchSetting : UDINT := 10;
	batchCount : UDINT;
	headCycleCount : UDINT;
	pressureBarOpenDelay : REAL;
	pressureBarCloseDelay : REAL;
	passthroughSetting : REAL := 5.0;
	passthroughOffset : REAL;
	passthroughPosition : REAL;
	lpaDwell : REAL;
	hpaDwell : REAL;
	sealBarDwell : REAL;
	sealBarTemperatureSetting : UDINT;
	sealBarTemperature : UDINT;
	sealFlattenersPosition : REAL;
	bagSkirtLength : REAL := 1.35;
	bagLength : REAL := 23.5;
	bagWidth : REAL := 17.5;
	bagThickness : REAL := 2.5;
	bagTensionSetting : REAL := 0.6;  // Bag takeup tension setting in amps
	bagDropTime : REAL;
	bagForwardSpeed : UDINT := 55;
	bagReverseSpeed : UDINT := 3;
	bagEdgePhotoeyeCovered : BOOL;
	printSpeed : UDINT := 6;
	printLength : REAL := 8.0;
	printOffset : REAL := 2.0;
	fillerCountSetting : UDINT;
	fillerCurrentCount : UDINT;
	fillerDropTime : REAL;
	loadPlateDelay : REAL;
	loadPlateDwell : REAL;
	exitConveyorDwell : REAL;
	vacuumDwell : REAL := 0.25;
	IBDDeflateDwellTime  : REAL := 0.75;
	IBDPackageEjectAssistDelayTime : REAL;
	IBDPackageEjectAssistDwellTime : REAL := 0.8;
	funnelInUse : BOOL;								// Funnel Enable/Disable
	funnelOpenDelay : REAL := 0.25;					// Funnel Open Delay after pressure bar open
	funnelOpeningTime : REAL := 0.5;				// For funnel w/o sensors only : Time required to consider funnel open after command to open
	funnelClosingTime : REAL := 0.5;				// For funnel w/o sensors only : Time required to consider funnel closed after command to close
	externalExitConveyorDwell : REAL;
	barcodeGoodReadCount : UDINT;
	barcodeBadReadCount : UDINT;
	barcodeBadReadFaultSetting : UDINT;
	barcodeStartPosition : REAL;
	barcodeScanDistance : REAL := 1.0;
	barcodeVerifierInUse : BOOL;
	barcodeLastReadString : STRING[100];
	lastCycleTime : REAL;
	averageCycleTime : REAL;
	resetAverageCycleTime : BOOL;
	bagOpenRetrySetting : INT := 3;
	bagOpenRetryCount : INT;
	bagOpenFeedNewBagSetting : INT := 1;
	bagOpenFeedNewBagCount : INT;
	currentJobID : INT;
	separateBeforeSeal : BOOL;
	activateDemoMode : BOOL;
	printerInUse : BOOL;
	printerInstalled : BOOL;
	lpaDuringBagFeedEnable : BOOL := TRUE;
	lpaBagEjectAssistEnable : BOOL := TRUE;

	(*Service Stuff*)
	lpaServiceOn : BOOL;
	lpaServiceOff : BOOL;
	lpaServicePulse : BOOL;
	hpaServiceOn :BOOL;
	hpaServicePulse : BOOL;
	exitConveyorStart : BOOL;
	exitConveyorStop : BOOL;
	exitConveyorJog : BOOL;
	exitConveyorJogTime : TIME;
	exitConveyorStartDwell : BOOL;
	pressureBarService : ServiceCommands;
	loadPlateService : ServiceCommands;
	forwardLoadPlateService : ServiceCommands;
	rearLoadPlateService : ServiceCommands;
	loadShelfService : ServiceCommands;
	IBDService : ServiceCommands;
	funnelService : ServiceCommands;
	baggerHeadService : ServiceCommands;
	jogBagForward : BOOL;
	jogBagReverse : BOOL;
	jogPassthroughForward : BOOL;
	jogPassthroughReverse : BOOL;
	sealBarServiceCycle : BOOL;
	sealBarServiceRetract : BOOL;
	sealBarServiceExtend : BOOL;
	bagOpenFingersServiceGrab : BOOL;
	bagOpenFingersServiceRelease : BOOL;
	sealFlattenersServiceRaise : BOOL;
	sealFlattenersServiceLower : BOOL;
	sealFlattenersServiceJogIn : BOOL;
	sealFlattenersServiceJogOut : BOOL;
	sealFlattenersManualPositionSetting : REAL;
	sealFlattenersMoveToManualPos : BOOL;
	passthroughManualPositionSetting : REAL;
	passthroughMoveToManualPos : BOOL;
	factoryTestMode : BOOL;
	vacuumServiceOn : BOOL;
	vacuumServiceOff : BOOL;
	printHeadServiceRaise : BOOL;
	printHeadServiceLower : BOOL;
	externalExitConveyorStart : BOOL;
	externalExitConveyorStop : BOOL;
	externalExitConveyorJog : BOOL;
	externalExitConveyorStartDwell : BOOL;
	triggerBarcodeReaderService : BOOL;
	
	(*Factoy Config*)
	bofSelection : BagOpenFingersSelection := BagOpenFingersSelection.PneumaticWithBagOpenSensors;
	sealFlattenersSelection : SealFlattenerSelection := SealFlattenerSelection.MotorizedSealFlatteners;
	printerSelection : LabelPrinterSelection := LabelPrinterSelection.ZebraPrinter203DPI;
	integratedExitConveyorSelection : IntegratedConveyorSelection := IntegratedConveyorSelection.RearExit;
	externalExitConveyorSelection : ExteralConveyorSelection := ExteralConveyorSelection.NotInstalled;
	packageEjectSelection : PackageEjectionSelection := PackageEjectionSelection.RearRetractingLoadPlate;
	independentBagDeflatorSelection : BagDeflatorSelection := BagDeflatorSelection.NotInstalled;
	cycleStartButtonSelection : PalmButtonSelection := PalmButtonSelection.DualPalmButton;
	barcodeVerifierSelection : BCVSelection := BCVSelection.NotInstalled;
	baggerModelSelection : ModelSelection;
	auxIOConfig : AuxIOConfiguration;
	fillerFactorySelection : FillerSelection;
	funnelFactorySelection : FunnelSelection;
	murrIOConfigVersion : CONFIG_VERSIONS := CONFIG_VERSIONS.V_1_3;
	printerConfigVersion : CONFIG_VERSIONS := CONFIG_VERSIONS.V_1_2;
	frontFilmFeedMotorConfigVersion : CONFIG_VERSIONS := CONFIG_VERSIONS.V_1_0;
	rearUnwindMotorConfigVersion : CONFIG_VERSIONS := CONFIG_VERSIONS.V_1_1;
	sealFlattenerMotorConfigVersion : CONFIG_VERSIONS := CONFIG_VERSIONS.V_1_0;
	
	(*Warnings*)
	printerRibbonLow : Warning;
	printerNotReady : Warning;
	waitingForPrinter : Warning;
	sealBarNotAtTemperature : Warning;
	recoveryModeActive : Warning;
	jobLoadRequired : Warning;
	baggerNotReady : Warning;
	demoModeIsActive : Warning;
	factoryTestModeActive : Warning;
	machineNotTested : Warning;
	packageEjectGuardRemoved : Warning;
	bagLevelLow : Warning;
	fillerModeCycleStartOnly : Warning;
	baggerInhibited : Warning;
	(*Misc*)
	pressureBarState : STRING;
    
    (*Counters*)
    baggerCycles : FB_CycleCounter;
	bagOpenFingerCycles : FB_CycleCounter;
	bagsMade : FB_CycleCounter;
	sealBarCycles : FB_CycleCounter;
	pressureBarCycles : FB_CycleCounter;
	passthroughChanges : FB_CycleCounter;
	loadPlateCycles : FB_CycleCounter;
	printerCycles : FB_CycleCounter;
	motorizedSealFlattenerCycles : FB_CycleCounter;
	bagOpenRetryTotal : FB_CycleCounter;
	bagsRejectedTotal : FB_CycleCounter;
	resettableBagsMade : FB_CycleCounter;
	
	(*Predictive Maint.*)
	airFilterClean : FB_PredictiveMaint := (target := 30000, count := 0, name := 'Clean Air Filter');
	driveRollerClean : FB_PredictiveMaint := (target := 20000, count := 0, name := 'Clean Drive Rollers', units := 'Inches of Bag');
	printHeadClean : FB_PredictiveMaint := (target := 10000, count := 0, name := 'Clean Print Head', units := 'Printer Cycles');
	pressureBarGuideShaftGuides : FB_PredictiveMaint := (target := 0, count := 127888, name := 'Replace Guide Shafts');
	
	pressureBarLeak : FB_CylinderLeak := (maximumStrokeTime := 5.0, name := 'Pressure Bar Stroke', units := 'Seconds');
	loadPlateLeak : FB_CylinderLeak := (maximumStrokeTime := 2.0, name := 'Load Plate Stroke', units := 'Seconds');
	
	msfHorizontalMotorTemp : FB_DriveTemp := (maxTemp := 60.0, name := 'MSF Motor Temp.', units := 'deg C');
	bagDeliveryMotorTemp : FB_DriveTemp := (maxTemp := 60.0, name := 'Bag Delivery Motor Temp.', units := 'deg C');
	passthroughMotorTemp : FB_DriveTemp := (maxTemp := 60.0, name := 'Passthrough Motor Temp.', units := 'deg C');
	
	(*Info*)
	faultActive : BOOL;

END_VAR

VAR_GLOBAL CONSTANT
	murrIOConfigVersionMax : CONFIG_VERSIONS := CONFIG_VERSIONS.V_1_3;
	printerConfigVersionMax : CONFIG_VERSIONS := CONFIG_VERSIONS.V_1_2;
	frontFilmFeedMotorConfigVersionMax : CONFIG_VERSIONS := CONFIG_VERSIONS.V_1_0;
	rearUnwindMotorConfigVersionMax : CONFIG_VERSIONS := CONFIG_VERSIONS.V_1_1;
	sealFlattenerMotorConfigVersionMax : CONFIG_VERSIONS := CONFIG_VERSIONS.V_1_0;
END_VAR

// Device/Application/ObjectHandling/GlobalObjects
{attribute 'qualified_only'}
{attribute 'global_init_slot' := '49995'}
VAR_GLOBAL CONSTANT
	MAX_OBJECTS : UINT := 750;
	MAX_CYLINDERS : UINT := 20;
	MAX_MOTORS : UINT := 10;
	MAX_FAULTS : UINT := 300;
	MAX_LOGS : UINT := 100;
	MAX_LOGGABLE : UINT := 500;
	MAX_EXECUTEABLE : UINT := 300;
END_VAR

VAR_GLOBAL
	CollectionOfAllObjects : FB_CollectionHandlerAll; 
	CollectionOfFaults : FB_CollectionHandlerFaults; 
// 	CollectionOfCylinders : FB_CollectionHandlerCylinders;
// 	CollectionOfPositionableMotors : FB_CollectionHandlerPositionableMotors;
	CollectionOfActiveFaults : FB_CollectionHandlerActiveFaults; 
	CollectionOfLogs : FB_CollectionHandlerLogs; 
	CollectionOfLoggable : FB_CollectionHandlerLoggable;
	CollectionOfExecutable : FB_CollectionHandlerExecutable;
	CollectionOfInitialzable : FB_CollectionHandlerInitializable;
END_VAR

// Device/Application/Globals
{attribute 'qualified_only'}
VAR_GLOBAL
    firstScan : BOOL; //First Scan Bit
    pressureBarServoCommsType : MODBUS_COMM_TYPE;  //Comm path to Pressure Bar Servo - 0 = TCP, 1 = RTU
    STEPS_PER_INCH : INT;  //Steps Per Inch for Pressure Bar Servos
    enableDryCycle : BOOL;          // Enable dry cycle
	SystemLog : FB_InternalLogger;
	jawMovingIn : BOOL;
	passthroughChangedFromJog : BOOL;
	machinePowerOK : BOOL;
END_VAR

VAR_GLOBAL CONSTANT
    STEPS_PER_INCH_SEAL_FLATTENER_HORIZONTAL_AXIS_MOTOR  : INT := 2500;
    STEPS_PER_INCH_SEAL_FLATTENER_VERTICAL_AXIS_MOTOR : INT := 2890;        //Steps per inch for NEMA 17 seal flattener finger motor
    STEPS_PER_INCH_BIG_MOTOR : INT := 21872;        //Steps per inch for NEMA 17 motor
    STEPS_PER_INCH_SMALL_MOTOR : INT := 19600;        //Steps per inch for NEMA 11 motor
    STEPS_PER_INCH_SHOW_MOTOR : INT := 18900;        //Steps per inch for NEMA 11 motor
    STEPS_PER_INCH_PRINTER : INT := 4498;            //Steps per inch for printer step servo
    STEPS_PER_INCH_20_DEGREE_BAG_DELIVERY : INT := 5093; // Steps per inch for 20 degree bag delivery motors
	STEPS_PER_INCH_PRO24_BAG_DELIVERY : INT := 4428; // Steps per inch for 20 degree bag delivery motors
	STEPS_PER_INCH_ADJUSTABLE_PASSTHROUGH : INT := 3030;  // Steps per inch for the Adjustable Passthrough motor
	STEPS_PER_INCH_TFBelt : INT := 3030;  // Steps per inch for the Adjustable Passthrough motor
	STEPS_PER_INCH_TFLS : INT := 10000;  // Steps per inch for the Adjustable Passthrough motor
    VELOCITY_IPS_MULTIPLIER_20_DEGREE_BAG_DELIVERY: REAL := 53;
    PASSTHROUGH_ZERO_OFFSET : REAL := 2;            //Zero offset for passthough (minimum passthough)
    MAX_BAG_WIDTH : REAL := 18;                //Passthrough setting
	AMP_MOTOR_RPI : INT := 10;
	MAX_LOGGED_ITEMS : UINT := 500;	// Max items to be logged
END_VAR

VAR_GLOBAL
    headCycleCount : DINT;                 // Head Cycle Counts
	headCycleCount2 : DINT;                 // Head Cycle Counts
    bagGrabberCycleCount : DINT;         // Bag Grabber Cycle Counts
    solenoidCycleCount1 : DINT;         // Solenoid Cycle Cycle Counts (first solenoid)
    motorizedSealFlattenersCount : DINT;         // MSF Cycle Counts
    bagOpenFingersCount : DINT;        // Bag Open Finger Cycles
    sealFlattenerFingersCount : DINT;  // Seal Flattener Fingers Cycle Count
    electricPressureBarCount : DINT;    // Electric Pressure bar Cycle count
    sealBarCount : DINT;                 // Seal bar Cycle count
    bagDeliveryCycleCount : DINT;        // Bag Delivery Cycle Count
    printerCycleCounts : DINT;            // Printer Cycle Counts
    bagsMadeCount : DINT;                // Bags Made
    passthroughChangeCount : DINT;        // Passthrough Changes
	passthroughChangeDistance : UDINT;	// Passthrough Distance Changes in .1 Inches
	solenoidCycleCount2 : DINT;     	// Solenoid Cycle Cycle Counts (Strech SX)	
	solenoidFailureCount2 : UDINT;		// Solenoid Failure Count (Strech SX)
	pickAndPlaceCycleCount : UDINT;		// Pick and place cycle count
	passthroughChangeCount2 : DINT;        // Passthrough Changes
	passthroughChangeDistance2 : UDINT;	// Passthrough Distance Changes in .1 Inches
	bagFailedToGrabBothFingersCount : UDINT; // Both Fingers failed to grab bag
	bagFailedToGrabRightFingerCount : UDINT; // Right Bag Open Finger Failed to Grab Bag
	bagFailedToGrabLeftFingerCount : UDINT; // Left Bag Open Finger Failed to Grab Bag
	successfulBagOpenCount : UDINT;			// Successful Bag Open Count
	rejectedBagCount : UDINT;				// Rejected bag count 
    dryCycleCount  :UDINT;                   // Dry cycle count
	lastPrinterDelta : TIME := T#100MS;
	factoryTestComplete : BOOL;		// 1000 bags test done
END_VAR

// Device/Application/Programs/PRG_MainProgram
PROGRAM PRG_MainProgram
VAR
    incrementSolenoidCounter1 : R_TRIG();
    incrementSolenoidCounter2 : R_TRIG();
    incrementSolenoidFailedCounter2 : R_TRIG();
    GripperCycleCount : DINT; //Gripper Cycle Counter
    runPrinterPB : BOOL;
    cycleTimeMax : TIME;
    cycleTimeMaxDINT : DINT;
    ctfb : OSCAT_BASIC.CYCLE_TIME();
    profileThis :BOOL;
    solenoidState1 : SOLENOID_TEST_STATES;
    solenoidState2 : SOLENOID_TEST_STATES;
    getTimeTilPMMI : TimeLeftFB();
	displayPassthroughChangeDistance : REAL;
	displayPassthroughChangeDistance2 : REAL;
	checkSolenoid2ExtendTimer : TON := (PT := T#100MS);
	checkedSolenoid2Status : BOOL;
	firstScanDone : BOOL;
	printDeltaTimer : TON := (PT := T#5S);
	lastPrinterDelta : TIME;
	endPrintOSF : Standard.R_TRIG;
	CSVWriter : FB_WriteToFile() := (xFilePath := 'C:/printerDelta.csv');
	stringToLog : STRING;
	testWrite : BOOL;
	hmiLight : FB_HMILight;
	versionInfo : VERSION;
	recipieManager : Recipe_Management.RecipeManCommands;
	recipeName : STRING;
	recResult : DWORD;
	testRead : BOOL;
	testCreate : BOOL;
	saveParametersTimer : Standard.TON := (PT := T#10M);
END_VAR

//    Program: Main (PLC_PRG)
//    Description: This program serves as a base for the MOAB Prototype
//    Created by: Ben Hess
//    Created Date: January 16th, 2018

printDeltaTimer(IN := oPrinterStartPrint);
saveParametersTimer(IN := NOT saveParametersTimer.Q);
IF saveParametersTimer.Q THEN
	recResult := recipieManager.GetRecipeNames('Recipes', ADR(recipeName),1,0);
	recResult := recipieManager.ReadAndSaveRecipe(RecipeDefinitionName := 'Recipes', RecipeName := recipeName);
	saveParametersTimer.IN := FALSE;
END_IF

IF testCreate THEN
// 	recResult := recipieManager.CreateRecipe(RecipeDefinitionName := 'Recipes', RecipeName := 'Automatic');
// 	recResult := recipieManager.ReadAndSaveRecipe(RecipeDefinitionName := 'Recipes', RecipeName := recipeName);
 	testCreate := FALSE;
	SaveValues();
END_IF

IF testRead THEN
// 	recResult := recipieManager.GetRecipeNames('Recipes', ADR(recipeName),1,0);
// 	recResult := recipieManager.LoadAndWriteRecipe(RecipeDefinitionName := 'Recipes', RecipeName := recipeName);
 	testRead := FALSE;
	RecallValues();
END_IF

// 
// CSVWriter(
// 	xFilePath:= , 
// 	xText_Write:= , 
// 	xAppend_OverWrite:= TRUE, 
// 	xAppend_Pos:= , 
// 	xWrite:= , 
// 	xRead:= , 
// 	xLine_No_To_Read:= , 
// 	xText_Read=> , 
// 	xDone=> );
// IF CSVWriter.xDone THEN
// 	CSVWriter.xWrite := FALSE;
// END_IF

ctfb(ct_max => cycleTimeMax);
cycleTimeMaxDINT := TIME_TO_DINT(cycleTimeMax);
profileThis := TIME_TO_DINT(ctfb.ct_last) >= 25;
// Run other programs
//PRG_PneumaticHead();
PRG_Bagger();
Faults();
versionInfo := GetVersion();
HMIData.version := Standard.CONCAT(TO_STRING(versionInfo.uiMajor),'.');
	BPLog.AppendToString(ADR(HMIData.version), CONCAT(TO_STRING(versionInfo.uiMinor),'.'));
	BPLog.AppendToString(ADR(HMIData.version), CONCAT(TO_STRING(versionInfo.uiServicePack),'.'));
	BPLog.AppendToString(ADR(HMIData.version), TO_STRING(versionInfo.uiPatch));
	BPLog.AppendToString(ADR(HMIData.version), TO_STRING(GetTextProperty("VersionPostfix")));
IF NOT firstScanDone THEN
	GlobalObjects.CollectionOfLoggable.RegisterAll(internalLogger := Globals.SystemLog);
	GlobalObjects.CollectionOfInitialzable.InitializeAll();
	firstScanDone := TRUE;
	// After first scan turn off flag set by StartDone system event
	Globals.firstScan := FALSE;	
END_IF

// Start executing objects that implement IExecuteAutomatically 
IF firstScanDone THEN
	GlobalObjects.CollectionOfExecutable.ExecuteAll();
	Globals.SystemLog();
END_IF




IF HMIData.ackAllFaults THEN
	GlobalObjects.CollectionOfActiveFaults.AckAll();
	HMIData.ackAllFaults := FALSE;
END_IF

getTimeTilPMMI(targetDate := DT#2018-10-14-8:0:0);


//First scan flag is set by task handler and reset in main routine here
IF Globals.firstScan THEN
    Globals.firstScan := FALSE;
END_IF

displayPassthroughChangeDistance := (UDINT_TO_REAL(Globals.passthroughChangeDistance) / 10);
displayPassthroughChangeDistance2 := (UDINT_TO_REAL(Globals.passthroughChangeDistance2) / 10.0);

END_PROGRAM

// Device/Application/SaveValues
FUNCTION SaveValues : DWORD
VAR
	recipieManager : Recipe_Management.RecipeManCommands;
	recipeName : STRING;
	recResult : DWORD;
END_VAR

recResult := recipieManager.CreateRecipe(RecipeDefinitionName := 'Recipes', RecipeName := 'Automatic');
recResult := recipieManager.GetRecipeNames('Recipes', ADR(recipeName),1,0);
recResult := recipieManager.ReadAndSaveRecipe(RecipeDefinitionName := 'Recipes', RecipeName := recipeName);

END_FUNCTION

